C03632=1040.909,-108.162,425.924,168.760,35.372,156.676
C03633=1040.915,-107.912,425.914,168.762,35.372,156.676
C03634=1040.921,-107.663,425.904,168.765,35.371,156.675
C03635=1040.927,-107.413,425.894,168.767,35.371,156.675
C03636=1040.934,-107.163,425.885,168.770,35.371,156.675
C03637=1040.940,-106.913,425.875,168.772,35.371,156.675
C03638=1040.945,-106.663,425.865,168.775,35.370,156.675
C03639=1040.952,-106.414,425.855,168.777,35.370,156.675
C03640=1040.958,-106.164,425.845,168.779,35.370,156.675
C03641=1040.964,-105.914,425.836,168.781,35.370,156.675
C03642=1040.970,-105.665,425.826,168.784,35.370,156.675
C03643=1040.976,-105.414,425.816,168.786,35.369,156.675
C03644=1040.982,-105.165,425.806,168.789,35.369,156.675
C03645=1040.988,-104.915,425.796,168.791,35.369,156.675
C03646=1040.994,-104.666,425.787,168.794,35.369,156.675
C03647=1041.000,-104.416,425.776,168.796,35.369,156.675
C03648=1041.006,-104.166,425.766,168.799,35.368,156.674
C03649=1041.013,-103.917,425.757,168.801,35.368,156.674
C03650=1041.019,-103.667,425.747,168.804,35.368,156.674
C03651=1041.024,-103.417,425.736,168.806,35.368,156.674
C03652=1041.031,-103.168,425.727,168.809,35.368,156.674
C03653=1041.037,-102.918,425.717,168.811,35.367,156.674
C03654=1041.043,-102.668,425.706,168.814,35.368,156.674
C03655=1041.049,-102.418,425.697,168.816,35.368,156.674
C03656=1041.055,-102.169,425.687,168.819,35.367,156.674
C03657=1041.061,-101.919,425.677,168.821,35.367,156.674
C03658=1041.067,-101.669,425.666,168.824,35.367,156.674
C03659=1041.074,-101.419,425.656,168.826,35.367,156.674
C03660=1041.080,-101.170,425.646,168.829,35.367,156.674
C03661=1041.086,-100.920,425.636,168.831,35.367,156.674
C03662=1041.092,-100.670,425.626,168.834,35.366,156.674
C03663=1041.098,-100.421,425.616,168.836,35.366,156.674
C03664=1041.105,-100.134,425.604,168.839,35.366,156.674
C03665=1041.112,-99.846,425.592,168.842,35.366,156.673
C03666=1041.120,-99.559,425.581,168.845,35.366,156.673
C03667=1041.127,-99.272,425.569,168.847,35.366,156.673
C03668=1041.133,-99.022,425.559,168.850,35.365,156.673
C03669=1041.139,-98.772,425.550,168.852,35.365,156.673
C03670=1041.145,-98.523,425.539,168.855,35.366,156.673
C03671=1041.151,-98.273,425.529,168.857,35.366,156.673
C03672=1041.157,-98.024,425.519,168.860,35.365,156.673
C03673=1041.163,-97.773,425.508,168.862,35.365,156.673
C03674=1041.170,-97.524,425.498,168.865,35.365,156.673
C03675=1041.175,-97.274,425.488,168.867,35.365,156.673
C03676=1041.182,-97.025,425.478,168.870,35.365,156.673
C03677=1041.187,-96.775,425.467,168.871,35.365,156.673
C03678=1041.194,-96.525,425.457,168.874,35.365,156.673
C03679=1041.199,-96.276,425.446,168.876,35.365,156.673
C03680=1041.206,-96.025,425.436,168.878,35.365,156.673
C03681=1041.212,-95.776,425.425,168.881,35.365,156.673
C03682=1041.218,-95.526,425.415,168.883,35.365,156.673
C03683=1041.224,-95.277,425.405,168.886,35.365,156.673
C03684=1041.230,-95.027,425.394,168.888,35.365,156.673
C03685=1041.236,-94.778,425.384,168.891,35.365,156.673
C03686=1041.242,-94.527,425.373,168.893,35.365,156.673
C03687=1041.248,-94.278,425.363,168.895,35.365,156.673
C03688=1041.254,-94.028,425.352,168.898,35.366,156.673
C03689=1041.260,-93.778,425.342,168.900,35.365,156.673
C03690=1041.266,-93.529,425.332,168.903,35.365,156.673
C03691=1041.272,-93.279,425.320,168.905,35.365,156.673
C03692=1041.279,-93.029,425.311,168.908,35.365,156.673
C03693=1041.284,-92.780,425.300,168.910,35.365,156.673
C03694=1041.290,-92.530,425.289,168.913,35.365,156.673
C03695=1041.297,-92.280,425.279,168.915,35.365,156.672
C03696=1041.303,-92.030,425.268,168.917,35.366,156.672
C03697=1041.309,-91.781,425.258,168.920,35.366,156.672
C03698=1041.315,-91.531,425.247,168.922,35.366,156.672
C03699=1041.321,-91.281,425.236,168.925,35.366,156.672
C03700=1041.327,-91.031,425.226,168.927,35.366,156.672
C03701=1041.333,-90.782,425.215,168.930,35.366,156.672
C03702=1041.340,-90.533,425.205,168.932,35.366,156.672
C03703=1041.346,-90.283,425.194,168.934,35.366,156.672
C03704=1041.351,-90.033,425.184,168.937,35.366,156.672
C03705=1041.358,-89.783,425.174,168.939,35.366,156.672
C03706=1041.364,-89.533,425.162,168.942,35.366,156.672
C03707=1041.370,-89.284,425.151,168.944,35.366,156.672
C03708=1041.376,-89.034,425.141,168.946,35.366,156.672
C03709=1041.382,-88.785,425.130,168.949,35.366,156.672
C03710=1041.389,-88.535,425.120,168.951,35.367,156.672
C03711=1041.395,-88.285,425.109,168.954,35.367,156.672
C03712=1041.400,-88.036,425.099,168.956,35.367,156.672
C03713=1041.407,-87.786,425.088,168.959,35.367,156.672
C03714=1041.413,-87.536,425.077,168.961,35.367,156.672
C03715=1041.419,-87.287,425.066,168.963,35.367,156.672
C03716=1041.426,-87.037,425.056,168.966,35.367,156.672
C03717=1041.432,-86.787,425.045,168.968,35.367,156.672
C03718=1041.438,-86.537,425.033,168.971,35.367,156.672
C03719=1041.445,-86.288,425.023,168.973,35.367,156.672
C03720=1041.450,-86.038,425.012,168.975,35.367,156.672
C03721=1041.456,-85.788,425.002,168.978,35.367,156.672
C03722=1041.463,-85.538,424.991,168.980,35.367,156.672
C03723=1041.469,-85.289,424.981,168.983,35.367,156.672
C03724=1041.475,-85.039,424.969,168.985,35.368,156.672
C03725=1041.481,-84.790,424.959,168.988,35.368,156.672
C03726=1041.488,-84.539,424.948,168.990,35.368,156.672
C03727=1041.493,-84.290,424.937,168.992,35.368,156.672
C03728=1041.501,-84.005,424.924,168.995,35.369,156.672
C03729=1041.508,-83.721,424.912,168.998,35.369,156.672
C03730=1041.515,-83.435,424.900,169.001,35.369,156.672
C03731=1041.522,-83.151,424.887,169.003,35.369,156.672
C03732=1041.529,-82.901,424.876,169.006,35.369,156.672
C03733=1041.535,-82.652,424.865,169.008,35.369,156.672
C03734=1041.541,-82.402,424.854,169.011,35.369,156.672
C03735=1041.547,-82.152,424.843,169.013,35.369,156.672
C03736=1041.554,-81.902,424.833,169.015,35.369,156.672
C03737=1041.560,-81.653,424.822,169.018,35.369,156.672
C03738=1041.566,-81.403,424.811,169.020,35.370,156.672
C03739=1041.573,-81.153,424.800,169.023,35.370,156.672
C03740=1041.579,-80.903,424.789,169.025,35.370,156.672
C03741=1041.585,-80.654,424.778,169.027,35.370,156.672
C03742=1041.591,-80.403,424.767,169.030,35.370,156.672
C03743=1041.598,-80.155,424.756,169.032,35.370,156.672
C03744=1041.604,-79.905,424.745,169.035,35.370,156.672
C03745=1041.610,-79.655,424.734,169.037,35.370,156.672
C03746=1041.616,-79.405,424.723,169.039,35.371,156.672
C03747=1041.622,-79.156,424.712,169.042,35.371,156.672
C03748=1041.628,-78.905,424.700,169.044,35.371,156.672
C03749=1041.634,-78.656,424.689,169.046,35.372,156.672
C03750=1041.642,-78.407,424.678,169.049,35.372,156.672
C03751=1041.647,-78.157,424.667,169.051,35.372,156.672
C03752=1041.654,-77.907,424.656,169.053,35.372,156.672
C03753=1041.660,-77.658,424.644,169.056,35.373,156.672
C03754=1041.666,-77.408,424.633,169.058,35.373,156.672
C03755=1041.672,-77.158,424.622,169.060,35.373,156.672
C03756=1041.678,-76.909,424.610,169.063,35.374,156.672
C03757=1041.684,-76.659,424.600,169.065,35.374,156.672
C03758=1041.690,-76.409,424.588,169.068,35.374,156.672
C03759=1041.696,-76.160,424.577,169.070,35.375,156.672
C03760=1041.703,-75.910,424.565,169.072,35.375,156.672
C03761=1041.709,-75.661,424.555,169.075,35.375,156.672
C03762=1041.715,-75.410,424.543,169.077,35.375,156.672
C03763=1041.722,-75.161,424.531,169.079,35.376,156.672
C03764=1041.727,-74.911,424.520,169.082,35.376,156.672
C03765=1041.734,-74.661,424.509,169.084,35.376,156.672
C03766=1041.740,-74.412,424.498,169.086,35.376,156.672
C03767=1041.746,-74.162,424.486,169.089,35.376,156.672
C03768=1041.752,-73.913,424.475,169.091,35.377,156.672
C03769=1041.758,-73.663,424.464,169.093,35.377,156.672
C03770=1041.765,-73.413,424.452,169.096,35.378,156.672
C03771=1041.771,-73.164,424.441,169.098,35.378,156.672
C03772=1041.776,-72.913,424.429,169.100,35.379,156.673
C03773=1041.782,-72.665,424.417,169.103,35.379,156.672
C03774=1041.789,-72.414,424.406,169.105,35.380,156.673
C03775=1041.795,-72.166,424.394,169.107,35.380,156.673
C03776=1041.800,-71.915,424.383,169.109,35.380,156.673
C03777=1041.807,-71.665,424.371,169.112,35.380,156.673
C03778=1041.813,-71.416,424.360,169.114,35.381,156.673
C03779=1041.820,-71.166,424.348,169.116,35.381,156.673
C03780=1041.825,-70.917,424.336,169.119,35.382,156.673
C03781=1041.831,-70.667,424.324,169.121,35.382,156.673
C03782=1041.837,-70.417,424.313,169.123,35.383,156.673
C03783=1041.844,-70.168,424.302,169.126,35.383,156.673
C03784=1041.850,-69.918,424.290,169.128,35.383,156.673
C03785=1041.855,-69.669,424.278,169.130,35.384,156.673
C03786=1041.862,-69.419,424.266,169.132,35.384,156.673
C03787=1041.868,-69.169,424.255,169.135,35.385,156.673
C03788=1041.874,-68.920,424.243,169.137,35.385,156.673
C03789=1041.880,-68.669,424.232,169.139,35.386,156.673
C03790=1041.886,-68.420,424.220,169.142,35.386,156.673
C03791=1041.893,-68.171,424.208,169.144,35.386,156.673
C03792=1041.899,-67.888,424.195,169.147,35.387,156.673
C03793=1041.907,-67.605,424.182,169.149,35.387,156.673
C03794=1041.914,-67.323,424.168,169.152,35.388,156.673
C03795=1041.920,-67.040,424.155,169.154,35.389,156.674
C03796=1041.926,-66.790,424.143,169.157,35.389,156.674
C03797=1041.933,-66.540,424.131,169.159,35.390,156.674
C03798=1041.939,-66.291,424.119,169.161,35.390,156.674
C03799=1041.945,-66.042,424.108,169.163,35.390,156.674
C03800=1041.951,-65.791,424.096,169.166,35.390,156.674
C03801=1041.957,-65.542,424.084,169.168,35.391,156.674
C03802=1041.964,-65.293,424.072,169.170,35.392,156.674
C03803=1041.969,-65.042,424.060,169.173,35.392,156.674
C03804=1041.976,-64.793,424.048,169.175,35.393,156.674
C03805=1041.982,-64.544,424.037,169.177,35.393,156.674
C03806=1041.989,-64.294,424.025,169.179,35.393,156.674
C03807=1041.994,-64.044,424.013,169.182,35.394,156.674
C03808=1042.001,-63.794,424.001,169.184,35.394,156.674
C03809=1042.007,-63.545,423.989,169.186,35.395,156.674
C03810=1042.013,-63.295,423.977,169.189,35.395,156.674
C03811=1042.019,-63.045,423.966,169.192,35.396,156.674
C03812=1042.026,-62.796,423.954,169.194,35.396,156.674
C03813=1042.031,-62.546,423.941,169.196,35.396,156.674
C03814=1042.038,-62.297,423.929,169.199,35.397,156.675
C03815=1042.044,-62.047,423.918,169.201,35.398,156.675
C03816=1042.050,-61.797,423.905,169.203,35.398,156.675
C03817=1042.057,-61.547,423.894,169.205,35.399,156.675
C03818=1042.063,-61.298,423.882,169.208,35.399,156.675
C03819=1042.069,-61.049,423.870,169.210,35.399,156.675
C03820=1042.075,-60.799,423.858,169.212,35.400,156.675
C03821=1042.082,-60.549,423.846,169.214,35.400,156.675
C03822=1042.088,-60.300,423.834,169.217,35.401,156.675
C03823=1042.094,-60.050,423.821,169.219,35.402,156.675
C03824=1042.100,-59.800,423.810,169.221,35.402,156.675
C03825=1042.107,-59.551,423.798,169.224,35.402,156.675
C03826=1042.113,-59.301,423.786,169.226,35.403,156.675
C03827=1042.119,-59.051,423.774,169.228,35.403,156.675
C03828=1042.126,-58.802,423.762,169.230,35.404,156.675
C03829=1042.132,-58.552,423.749,169.233,35.405,156.675
C03830=1042.139,-58.302,423.737,169.235,35.405,156.675
C03831=1042.144,-58.053,423.725,169.237,35.405,156.675
C03832=1042.150,-57.804,423.713,169.239,35.406,156.676
C03833=1042.157,-57.554,423.701,169.242,35.406,156.676
C03834=1042.163,-57.304,423.689,169.244,35.407,156.676
C03835=1042.170,-57.055,423.677,169.246,35.407,156.676
C03836=1042.176,-56.805,423.665,169.248,35.408,156.676
C03837=1042.182,-56.555,423.652,169.251,35.408,156.676
C03838=1042.189,-56.306,423.640,169.253,35.409,156.676
C03839=1042.196,-56.056,423.628,169.255,35.409,156.676
C03840=1042.201,-55.806,423.616,169.257,35.410,156.676
C03841=1042.208,-55.556,423.604,169.260,35.410,156.676
C03842=1042.214,-55.308,423.592,169.262,35.410,156.676
C03843=1042.220,-55.058,423.580,169.264,35.411,156.676
C03844=1042.227,-54.808,423.568,169.266,35.412,156.676
C03845=1042.233,-54.558,423.555,169.269,35.412,156.676
C03846=1042.239,-54.309,423.543,169.271,35.413,156.676
C03847=1042.246,-54.059,423.531,169.273,35.413,156.676
C03848=1042.252,-53.809,423.519,169.275,35.414,156.677
C03849=1042.259,-53.560,423.506,169.278,35.414,156.677
C03850=1042.265,-53.310,423.493,169.280,35.415,156.677
C03851=1042.271,-53.061,423.481,169.282,35.416,156.677
C03852=1042.278,-52.811,423.469,169.284,35.416,156.677
C03853=1042.284,-52.561,423.457,169.286,35.416,156.677
C03854=1042.291,-52.312,423.445,169.289,35.417,156.677
C03855=1042.296,-52.062,423.432,169.291,35.417,156.677
C03856=1042.305,-51.781,423.419,169.293,35.418,156.677
C03857=1042.312,-51.499,423.404,169.297,35.419,156.677
C03858=1042.318,-51.218,423.391,169.299,35.419,156.677
C03859=1042.326,-50.937,423.376,169.302,35.420,156.677
C03860=1042.332,-50.687,423.364,169.304,35.420,156.677
C03861=1042.338,-50.437,423.352,169.306,35.421,156.677
C03862=1042.345,-50.188,423.340,169.309,35.421,156.677
C03863=1042.351,-49.938,423.327,169.311,35.422,156.678
C03864=1042.357,-49.688,423.314,169.313,35.423,156.678
C03865=1042.364,-49.439,423.302,169.315,35.424,156.678
C03866=1042.370,-49.189,423.290,169.317,35.424,156.678
C03867=1042.376,-48.940,423.276,169.319,35.425,156.678
C03868=1042.382,-48.690,423.264,169.322,35.426,156.678
C03869=1042.388,-48.440,423.252,169.324,35.426,156.678
C03870=1042.395,-48.191,423.239,169.326,35.427,156.678
C03871=1042.400,-47.941,423.226,169.328,35.428,156.678
C03872=1042.407,-47.692,423.213,169.330,35.428,156.678
C03873=1042.413,-47.442,423.201,169.333,35.429,156.679
C03874=1042.419,-47.192,423.188,169.335,35.430,156.679
C03875=1042.425,-46.943,423.175,169.337,35.431,156.679
C03876=1042.431,-46.693,423.162,169.339,35.431,156.679
C03877=1042.438,-46.444,423.150,169.341,35.432,156.679
C03878=1042.445,-46.194,423.137,169.343,35.433,156.679
C03879=1042.451,-45.944,423.124,169.346,35.433,156.679
C03880=1042.457,-45.695,423.111,169.348,35.434,156.679
C03881=1042.463,-45.445,423.098,169.350,35.435,156.679
C03882=1042.469,-45.195,423.086,169.352,35.435,156.679
C03883=1042.476,-44.946,423.073,169.354,35.436,156.679
C03884=1042.482,-44.696,423.061,169.356,35.436,156.680
C03885=1042.488,-44.447,423.047,169.359,35.437,156.680
C03886=1042.494,-44.197,423.035,169.362,35.438,156.680
C03887=1042.501,-43.948,423.022,169.364,35.438,156.680
C03888=1042.507,-43.698,423.010,169.366,35.439,156.680
C03889=1042.513,-43.449,422.996,169.368,35.440,156.680
C03890=1042.519,-43.198,422.983,169.370,35.440,156.680
C03891=1042.526,-42.949,422.971,169.372,35.441,156.680
C03892=1042.532,-42.699,422.958,169.375,35.442,156.680
C03893=1042.538,-42.450,422.945,169.377,35.443,156.680
C03894=1042.544,-42.200,422.932,169.379,35.443,156.681
C03895=1042.551,-41.951,422.920,169.381,35.444,156.681
C03896=1042.557,-41.701,422.907,169.383,35.445,156.681
C03897=1042.564,-41.451,422.893,169.385,35.445,156.681
C03898=1042.570,-41.202,422.880,169.387,35.446,156.681
C03899=1042.576,-40.952,422.868,169.390,35.447,156.681
C03900=1042.582,-40.703,422.854,169.392,35.447,156.681
C03901=1042.589,-40.453,422.842,169.394,35.448,156.681
C03902=1042.595,-40.204,422.829,169.396,35.449,156.681
C03903=1042.602,-39.954,422.815,169.398,35.450,156.682
C03904=1042.608,-39.704,422.803,169.400,35.451,156.682
C03905=1042.614,-39.455,422.790,169.402,35.452,156.682
C03906=1042.621,-39.205,422.778,169.405,35.452,156.682
C03907=1042.627,-38.956,422.764,169.407,35.453,156.682
C03908=1042.634,-38.706,422.751,169.409,35.454,156.682
C03909=1042.640,-38.456,422.738,169.411,35.454,156.682
C03910=1042.646,-38.207,422.725,169.414,35.455,156.682
C03911=1042.652,-37.958,422.712,169.416,35.456,156.682
C03912=1042.658,-37.708,422.699,169.418,35.456,156.682
C03913=1042.665,-37.458,422.686,169.420,35.458,156.683
C03914=1042.671,-37.209,422.672,169.423,35.459,156.683
C03915=1042.677,-36.959,422.659,169.425,35.459,156.683
C03916=1042.683,-36.710,422.646,169.427,35.460,156.683
C03917=1042.689,-36.460,422.633,169.429,35.461,156.683
C03918=1042.695,-36.210,422.619,169.431,35.461,156.683
C03919=1042.702,-35.961,422.606,169.433,35.463,156.683
C03920=1042.708,-35.680,422.592,169.435,35.463,156.683
C03921=1042.716,-35.399,422.576,169.438,35.464,156.684
C03922=1042.723,-35.118,422.561,169.440,35.465,156.684
C03923=1042.730,-34.837,422.547,169.442,35.466,156.684
C03924=1042.737,-34.587,422.533,169.445,35.467,156.684
C03925=1042.743,-34.338,422.520,169.447,35.467,156.684
C03926=1042.749,-34.088,422.507,169.449,35.469,156.684
C03927=1042.755,-33.839,422.494,169.451,35.469,156.684
C03928=1042.762,-33.589,422.480,169.453,35.470,156.684
C03929=1042.767,-33.340,422.466,169.455,35.471,156.685
C03930=1042.773,-33.090,422.453,169.458,35.472,156.685
C03931=1042.780,-32.840,422.440,169.460,35.473,156.685
C03932=1042.786,-32.591,422.426,169.462,35.474,156.685
C03933=1042.792,-32.341,422.414,169.464,35.474,156.685
C03934=1042.799,-32.092,422.400,169.466,35.475,156.685
C03935=1042.805,-31.842,422.387,169.469,35.476,156.685
C03936=1042.812,-31.593,422.374,169.471,35.477,156.686
C03937=1042.818,-31.343,422.360,169.473,35.478,156.686
C03938=1042.825,-31.093,422.347,169.475,35.478,156.686
C03939=1042.831,-30.844,422.333,169.477,35.479,156.686
C03940=1042.836,-30.595,422.319,169.479,35.480,156.686
C03941=1042.843,-30.345,422.306,169.481,35.481,156.686
C03942=1042.849,-30.095,422.293,169.483,35.482,156.686
C03943=1042.856,-29.846,422.279,169.485,35.483,156.686
C03944=1042.862,-29.596,422.266,169.487,35.483,156.686
C03945=1042.869,-29.347,422.252,169.489,35.484,156.687
C03946=1042.875,-29.098,422.239,169.491,35.485,156.687
C03947=1042.882,-28.848,422.225,169.493,35.486,156.687
C03948=1042.888,-28.598,422.212,169.495,35.487,156.687
C03949=1042.894,-28.348,422.198,169.498,35.487,156.687
C03950=1042.900,-28.099,422.185,169.501,35.489,156.687
C03951=1042.906,-27.850,422.171,169.503,35.489,156.687
C03952=1042.913,-27.600,422.158,169.505,35.490,156.687
C03953=1042.919,-27.350,422.145,169.507,35.491,156.688
C03954=1042.926,-27.100,422.131,169.509,35.491,156.688
C03955=1042.932,-26.851,422.118,169.511,35.493,156.688
C03956=1042.938,-26.602,422.104,169.513,35.493,156.688
C03957=1042.945,-26.352,422.090,169.515,35.494,156.688
C03958=1042.951,-26.102,422.077,169.517,35.495,156.688
C03959=1042.957,-25.853,422.062,169.519,35.496,156.688
C03960=1042.964,-25.603,422.049,169.521,35.497,156.689
C03961=1042.969,-25.354,422.035,169.523,35.498,156.689
C03962=1042.976,-25.104,422.021,169.525,35.499,156.689
C03963=1042.982,-24.855,422.008,169.527,35.500,156.689
C03964=1042.988,-24.605,421.994,169.529,35.501,156.689
C03965=1042.995,-24.356,421.980,169.531,35.502,156.689
C03966=1043.001,-24.106,421.966,169.533,35.503,156.689
C03967=1043.007,-23.856,421.952,169.536,35.504,156.690
C03968=1043.013,-23.607,421.939,169.538,35.505,156.690
C03969=1043.019,-23.358,421.926,169.540,35.506,156.690
C03970=1043.026,-23.108,421.911,169.542,35.506,156.690
C03971=1043.032,-22.859,421.897,169.544,35.508,156.690
C03972=1043.038,-22.608,421.883,169.546,35.508,156.690
C03973=1043.044,-22.359,421.870,169.548,35.510,156.691
C03974=1043.051,-22.110,421.856,169.550,35.510,156.691
C03975=1043.057,-21.860,421.842,169.552,35.511,156.691
C03976=1043.064,-21.610,421.828,169.554,35.512,156.691
C03977=1043.069,-21.361,421.814,169.556,35.513,156.691
C03978=1043.076,-21.112,421.800,169.558,35.514,156.691
C03979=1043.082,-20.862,421.787,169.560,35.515,156.691
C03980=1043.088,-20.612,421.773,169.562,35.516,156.691
C03981=1043.095,-20.363,421.758,169.564,35.517,156.692
C03982=1043.101,-20.114,421.745,169.566,35.518,156.692
C03983=1043.107,-19.864,421.731,169.569,35.519,156.692
C03984=1043.115,-19.582,421.715,169.572,35.520,156.692
C03985=1043.122,-19.301,421.699,169.574,35.521,156.692
C03986=1043.129,-19.018,421.684,169.576,35.522,156.692
C03987=1043.136,-18.737,421.668,169.579,35.523,156.693
C03988=1043.142,-18.487,421.654,169.581,35.524,156.693
C03989=1043.149,-18.238,421.640,169.583,35.525,156.693
C03990=1043.155,-17.988,421.626,169.585,35.526,156.693
C03991=1043.162,-17.739,421.611,169.586,35.527,156.693
C03992=1043.168,-17.489,421.598,169.588,35.528,156.693
C03993=1043.174,-17.239,421.584,169.590,35.529,156.693
C03994=1043.181,-16.990,421.570,169.592,35.530,156.694
C03995=1043.187,-16.740,421.556,169.594,35.531,156.694
C03996=1043.193,-16.491,421.541,169.596,35.531,156.694
C03997=1043.200,-16.241,421.528,169.598,35.533,156.694
C03998=1043.206,-15.993,421.513,169.600,35.533,156.694
C03999=1043.213,-15.743,421.500,169.603,35.535,156.694
C04000=1043.219,-15.492,421.485,169.605,35.535,156.695
C04001=1043.225,-15.244,421.471,169.607,35.536,156.695
C04002=1043.231,-14.993,421.457,169.609,35.537,156.695
C04003=1043.238,-14.745,421.443,169.611,35.539,156.695
C04004=1043.244,-14.495,421.428,169.613,35.539,156.695
C04005=1043.250,-14.245,421.414,169.615,35.541,156.695
C04006=1043.257,-13.996,421.400,169.617,35.541,156.695
C04007=1043.263,-13.746,421.386,169.619,35.543,156.696
C04008=1043.269,-13.497,421.371,169.621,35.543,156.696
C04009=1043.275,-13.247,421.358,169.623,35.545,156.696
C04010=1043.281,-12.998,421.343,169.625,35.545,156.696
C04011=1043.288,-12.748,421.328,169.627,35.547,156.696
C04012=1043.294,-12.498,421.314,169.629,35.548,156.697
C04013=1043.300,-12.249,421.300,169.631,35.549,156.697
C04014=1043.306,-11.999,421.286,169.634,35.550,156.697
C04015=1043.313,-11.750,421.272,169.636,35.551,156.697
C04016=1043.319,-11.501,421.257,169.638,35.552,156.697
C04017=1043.325,-11.251,421.242,169.640,35.553,156.697
C04018=1043.332,-11.002,421.228,169.642,35.554,156.698
C04019=1043.338,-10.752,421.213,169.644,35.555,156.698
C04020=1043.344,-10.503,421.200,169.646,35.556,156.698
C04021=1043.351,-10.253,421.185,169.647,35.557,156.698
C04022=1043.357,-10.004,421.170,169.649,35.558,156.698
C04023=1043.363,-9.754,421.156,169.651,35.559,156.698
C04024=1043.369,-9.504,421.141,169.653,35.560,156.698
C04025=1043.376,-9.255,421.127,169.655,35.561,156.699
C04026=1043.382,-9.006,421.113,169.657,35.562,156.699
C04027=1043.388,-8.756,421.098,169.660,35.563,156.699
C04028=1043.395,-8.507,421.084,169.662,35.564,156.699
C04029=1043.401,-8.258,421.069,169.664,35.565,156.699
C04030=1043.407,-8.007,421.055,169.666,35.567,156.700
C04031=1043.414,-7.758,421.041,169.668,35.567,156.700
C04032=1043.420,-7.509,421.026,169.670,35.569,156.700
C04033=1043.426,-7.259,421.011,169.672,35.569,156.700
C04034=1043.432,-7.009,420.997,169.674,35.571,156.700
C04035=1043.439,-6.760,420.983,169.676,35.571,156.700
C04036=1043.445,-6.511,420.968,169.678,35.573,156.701
C04037=1043.452,-6.261,420.953,169.679,35.574,156.701
C04038=1043.459,-6.012,420.939,169.681,35.575,156.701
C04039=1043.464,-5.762,420.925,169.683,35.576,156.701
C04040=1043.471,-5.513,420.910,169.685,35.577,156.701
C04041=1043.477,-5.263,420.895,169.688,35.578,156.701
C04042=1043.484,-5.014,420.881,169.690,35.579,156.701
C04043=1043.490,-4.765,420.866,169.692,35.580,156.702
C04044=1043.496,-4.515,420.851,169.694,35.581,156.702
C04045=1043.502,-4.265,420.837,169.696,35.582,156.702
C04046=1043.509,-4.015,420.823,169.698,35.583,156.702
C04047=1043.515,-3.766,420.808,169.700,35.584,156.702
C04048=1043.523,-3.483,420.791,169.702,35.585,156.703
C04049=1043.530,-3.199,420.774,169.704,35.587,156.703
C04050=1043.537,-2.915,420.757,169.706,35.588,156.703
C04051=1043.544,-2.633,420.740,169.708,35.589,156.703
C04052=1043.550,-2.384,420.726,169.710,35.590,156.703
C04053=1043.556,-2.134,420.711,169.712,35.591,156.704
C04054=1043.563,-1.884,420.696,169.715,35.592,156.704
C04055=1043.569,-1.635,420.681,169.717,35.594,156.704
C04056=1043.575,-1.386,420.666,169.719,35.595,156.704
C04057=1043.581,-1.136,420.651,169.721,35.596,156.704
C04058=1043.587,-0.886,420.636,169.722,35.597,156.705
C04059=1043.594,-0.637,420.621,169.724,35.598,156.705
C04060=1043.600,-0.388,420.607,169.726,35.600,156.705
C04061=1043.606,-0.138,420.592,169.728,35.600,156.705
C04062=1043.612,0.111,420.577,169.730,35.602,156.705
C04063=1043.619,0.361,420.562,169.732,35.603,156.706
C04064=1043.624,0.610,420.547,169.734,35.604,156.706
C04065=1043.630,0.860,420.532,169.736,35.605,156.706
C04066=1043.637,1.110,420.517,169.738,35.606,156.706
C04067=1043.643,1.359,420.502,169.740,35.608,156.706
C04068=1043.649,1.609,420.487,169.742,35.609,156.706
C04069=1043.655,1.858,420.472,169.744,35.610,156.707
C04070=1043.662,2.107,420.457,169.746,35.611,156.707
C04071=1043.668,2.357,420.442,169.748,35.612,156.707
C04072=1043.675,2.606,420.427,169.750,35.614,156.707
C04073=1043.681,2.856,420.412,169.751,35.614,156.707
C04074=1043.687,3.106,420.397,169.753,35.616,156.708
C04075=1043.693,3.355,420.382,169.755,35.617,156.708
C04076=1043.700,3.604,420.367,169.757,35.618,156.708
C04077=1043.706,3.853,420.352,169.760,35.619,156.708
C04078=1043.713,4.103,420.337,169.762,35.620,156.708
C04079=1043.718,4.353,420.321,169.764,35.621,156.709
C04080=1043.725,4.603,420.306,169.765,35.623,156.709
C04081=1043.731,4.852,420.291,169.767,35.623,156.709
C04082=1043.737,5.101,420.276,169.769,35.625,156.709
C04083=1043.744,5.350,420.261,169.771,35.626,156.709
C04084=1043.750,5.600,420.246,169.773,35.627,156.710
C04085=1043.756,5.850,420.231,169.775,35.628,156.710
C04086=1043.763,6.099,420.216,169.777,35.629,156.710
C04087=1043.769,6.348,420.201,169.778,35.631,156.710
C04088=1043.776,6.598,420.186,169.780,35.632,156.710
C04089=1043.781,6.848,420.170,169.783,35.633,156.710
C04090=1043.788,7.098,420.155,169.785,35.634,156.711
C04091=1043.794,7.346,420.140,169.787,35.635,156.711
C04092=1043.800,7.596,420.125,169.789,35.637,156.711
C04093=1043.807,7.845,420.110,169.791,35.637,156.711
C04094=1043.813,8.094,420.094,169.792,35.639,156.711
C04095=1043.820,8.344,420.079,169.794,35.640,156.712
C04096=1043.826,8.594,420.064,169.796,35.641,156.712
C04097=1043.833,8.843,420.049,169.798,35.642,156.712
C04098=1043.838,9.093,420.033,169.800,35.643,156.712
C04099=1043.845,9.342,420.018,169.802,35.644,156.712
C04100=1043.851,9.591,420.003,169.804,35.646,156.713
C04101=1043.858,9.841,419.988,169.806,35.646,156.713
C04102=1043.864,10.091,419.973,169.808,35.648,156.713
C04103=1043.871,10.340,419.957,169.810,35.649,156.713
C04104=1043.877,10.589,419.942,169.812,35.650,156.713
C04105=1043.884,10.839,419.927,169.814,35.651,156.714
C04106=1043.890,11.088,419.911,169.816,35.652,156.714
C04107=1043.896,11.338,419.896,169.817,35.654,156.714
C04108=1043.903,11.587,419.880,169.819,35.655,156.714
C04109=1043.909,11.837,419.865,169.821,35.656,156.714
C04110=1043.915,12.086,419.850,169.823,35.657,156.714
C04111=1043.922,12.335,419.835,169.825,35.658,156.715
C04112=1043.930,12.620,419.817,169.828,35.660,156.715
C04113=1043.937,12.906,419.800,169.830,35.661,156.715
C04114=1043.944,13.191,419.783,169.832,35.662,156.715
C04115=1043.951,13.476,419.765,169.834,35.663,156.716
C04116=1043.957,13.725,419.749,169.836,35.664,156.716
C04117=1043.964,13.975,419.734,169.838,35.665,156.716
C04118=1043.970,14.224,419.718,169.840,35.667,156.716
C04119=1043.976,14.474,419.703,169.841,35.668,156.716
C04120=1043.983,14.723,419.687,169.843,35.669,156.717
C04121=1043.989,14.973,419.672,169.845,35.671,156.717
C04122=1043.995,15.222,419.656,169.848,35.672,156.717
C04123=1044.001,15.472,419.641,169.850,35.673,156.717
C04124=1044.008,15.721,419.625,169.851,35.674,156.717
C04125=1044.014,15.971,419.609,169.853,35.675,156.718
C04126=1044.021,16.221,419.594,169.855,35.677,156.718
C04127=1044.027,16.470,419.577,169.857,35.678,156.718
C04128=1044.033,16.720,419.563,169.859,35.679,156.718
C04129=1044.040,16.969,419.547,169.860,35.680,156.718
C04130=1044.046,17.219,419.531,169.862,35.682,156.719
C04131=1044.052,17.468,419.516,169.864,35.682,156.719
C04132=1044.058,17.717,419.499,169.866,35.684,156.719
C04133=1044.065,17.967,419.484,169.869,35.685,156.719
C04134=1044.072,18.216,419.469,169.870,35.686,156.719
C04135=1044.077,18.465,419.453,169.872,35.688,156.720
C04136=1044.084,18.715,419.438,169.874,35.689,156.720
C04137=1044.090,18.964,419.421,169.876,35.690,156.720
C04138=1044.096,19.213,419.406,169.878,35.691,156.720
C04139=1044.103,19.463,419.391,169.879,35.692,156.720
C04140=1044.109,19.712,419.374,169.881,35.694,156.721
C04141=1044.116,19.962,419.358,169.883,35.695,156.721
C04142=1044.122,20.211,419.342,169.885,35.696,156.721
C04143=1044.128,20.461,419.327,169.887,35.697,156.721
C04144=1044.134,20.710,419.311,169.889,35.699,156.722
C04145=1044.141,20.959,419.295,169.891,35.700,156.722
C04146=1044.147,21.208,419.279,169.893,35.701,156.722
C04147=1044.153,21.458,419.264,169.895,35.703,156.722
C04148=1044.159,21.707,419.248,169.896,35.704,156.722
C04149=1044.165,21.957,419.232,169.898,35.705,156.723
C04150=1044.172,22.206,419.216,169.900,35.706,156.723
C04151=1044.178,22.457,419.200,169.902,35.707,156.723
C04152=1044.185,22.706,419.184,169.904,35.708,156.723
C04153=1044.191,22.955,419.168,169.905,35.710,156.723
C04154=1044.198,23.204,419.152,169.908,35.711,156.724
C04155=1044.204,23.453,419.136,169.910,35.712,156.724
C04156=1044.209,23.703,419.120,169.912,35.714,156.724
C04157=1044.216,23.952,419.105,169.913,35.715,156.724
C04158=1044.222,24.202,419.089,169.915,35.716,156.725
C04159=1044.229,24.451,419.073,169.917,35.718,156.725
C04160=1044.235,24.701,419.056,169.919,35.719,156.725
C04161=1044.242,24.950,419.041,169.920,35.720,156.725
C04162=1044.248,25.199,419.025,169.922,35.721,156.725
C04163=1044.254,25.448,419.008,169.924,35.723,156.726
C04164=1044.260,25.698,418.993,169.927,35.723,156.726
C04165=1044.267,25.948,418.977,169.929,35.725,156.726
C04166=1044.273,26.197,418.961,169.930,35.726,156.726
C04167=1044.279,26.447,418.945,169.932,35.727,156.726
C04168=1044.286,26.696,418.929,169.934,35.729,156.727
C04169=1044.292,26.945,418.913,169.936,35.730,156.727
C04170=1044.298,27.195,418.896,169.937,35.731,156.727
C04171=1044.305,27.444,418.881,169.939,35.732,156.727
C04172=1044.311,27.693,418.864,169.941,35.734,156.728
C04173=1044.317,27.943,418.848,169.943,35.735,156.728
C04174=1044.324,28.192,418.832,169.945,35.736,156.728
C04175=1044.330,28.442,418.816,169.947,35.738,156.728
C04176=1044.338,28.728,418.797,169.949,35.739,156.729
C04177=1044.345,29.015,418.779,169.951,35.741,156.729
C04178=1044.351,29.302,418.760,169.953,35.742,156.729
C04179=1044.359,29.588,418.741,169.955,35.744,156.729
C04180=1044.365,29.837,418.725,169.957,35.745,156.730
C04181=1044.371,30.086,418.709,169.959,35.746,156.730
C04182=1044.378,30.336,418.693,169.960,35.747,156.730
C04183=1044.384,30.586,418.677,169.963,35.749,156.730
C04184=1044.390,30.835,418.660,169.965,35.750,156.730
C04185=1044.396,31.084,418.644,169.967,35.751,156.731
C04186=1044.402,31.334,418.627,169.968,35.753,156.731
C04187=1044.409,31.583,418.611,169.970,35.754,156.731
C04188=1044.415,31.832,418.595,169.972,35.755,156.731
C04189=1044.421,32.081,418.579,169.973,35.756,156.732
C04190=1044.428,32.331,418.562,169.975,35.758,156.732
C04191=1044.434,32.581,418.546,169.977,35.759,156.732
C04192=1044.440,32.830,418.530,169.980,35.760,156.732
C04193=1044.446,33.079,418.514,169.981,35.762,156.732
C04194=1044.453,33.329,418.496,169.983,35.764,156.733
C04195=1044.459,33.578,418.480,169.985,35.765,156.733
C04196=1044.465,33.827,418.464,169.987,35.766,156.733
C04197=1044.471,34.077,418.448,169.988,35.767,156.733
C04198=1044.478,34.326,418.432,169.990,35.769,156.734
C04199=1044.484,34.576,418.415,169.992,35.770,156.734
C04200=1044.491,34.824,418.398,169.994,35.771,156.734
C04201=1044.497,35.075,418.382,169.996,35.773,156.734
C04202=1044.503,35.324,418.365,169.998,35.774,156.735
C04203=1044.509,35.573,418.349,170.000,35.775,156.735
C04204=1044.517,35.822,418.332,170.002,35.776,156.735
C04205=1044.523,36.072,418.316,170.003,35.778,156.735
C04206=1044.529,36.321,418.300,170.005,35.779,156.735
C04207=1044.535,36.571,418.283,170.007,35.780,156.736
C04208=1044.541,36.820,418.266,170.008,35.782,156.736
C04209=1044.547,37.069,418.250,170.010,35.783,156.736
C04210=1044.555,37.319,418.234,170.013,35.784,156.736
C04211=1044.561,37.568,418.218,170.015,35.786,156.737
C04212=1044.567,37.817,418.201,170.016,35.787,156.737
C04213=1044.573,38.067,418.184,170.018,35.788,156.737
C04214=1044.580,38.316,418.167,170.020,35.789,156.737
C04215=1044.586,38.565,418.151,170.021,35.791,156.738
C04216=1044.592,38.815,418.134,170.023,35.792,156.738
C04217=1044.598,39.064,418.117,170.025,35.793,156.738
C04218=1044.604,39.314,418.101,170.027,35.795,156.738
C04219=1044.610,39.564,418.084,170.029,35.796,156.739
C04220=1044.616,39.812,418.067,170.031,35.798,156.739
C04221=1044.622,40.062,418.051,170.033,35.799,156.739
C04222=1044.629,40.311,418.033,170.034,35.800,156.739
C04223=1044.635,40.560,418.017,170.036,35.802,156.739
C04224=1044.641,40.810,418.001,170.038,35.803,156.740
C04225=1044.648,41.059,417.984,170.040,35.804,156.740
C04226=1044.654,41.309,417.967,170.041,35.805,156.740
C04227=1044.661,41.558,417.950,170.043,35.807,156.740
C04228=1044.667,41.807,417.934,170.046,35.808,156.741
C04229=1044.673,42.056,417.917,170.047,35.810,156.741
C04230=1044.680,42.306,417.900,170.049,35.811,156.741
C04231=1044.686,42.555,417.883,170.051,35.813,156.741
C04232=1044.692,42.804,417.867,170.052,35.814,156.742
C04233=1044.698,43.054,417.849,170.054,35.815,156.742
C04234=1044.704,43.303,417.833,170.056,35.816,156.742
C04235=1044.711,43.553,417.815,170.058,35.818,156.742
C04236=1044.717,43.802,417.799,170.059,35.819,156.742
C04237=1044.723,44.051,417.782,170.062,35.821,156.743
C04238=1044.729,44.301,417.765,170.064,35.822,156.743
C04239=1044.735,44.550,417.748,170.065,35.823,156.743
C04240=1044.742,44.836,417.729,170.067,35.825,156.744
C04241=1044.749,45.123,417.708,170.069,35.827,156.744
C04242=1044.756,45.410,417.689,170.071,35.829,156.744
C04243=1044.763,45.696,417.670,170.073,35.830,156.744
C04244=1044.769,45.946,417.653,170.076,35.832,156.745
C04245=1044.776,46.194,417.636,170.077,35.833,156.745
C04246=1044.782,46.444,417.619,170.079,35.834,156.745
C04247=1044.788,46.693,417.601,170.081,35.836,156.745
C04248=1044.794,46.942,417.584,170.082,35.837,156.746
C04249=1044.801,47.192,417.568,170.084,35.839,156.746
C04250=1044.806,47.441,417.550,170.086,35.840,156.746
C04251=1044.813,47.691,417.533,170.087,35.841,156.746
C04252=1044.819,47.940,417.517,170.089,35.843,156.747
C04253=1044.825,48.190,417.499,170.092,35.844,156.747
C04254=1044.831,48.439,417.482,170.093,35.846,156.747
C04255=1044.838,48.689,417.465,170.095,35.847,156.747
C04256=1044.843,48.938,417.448,170.097,35.848,156.748
C04257=1044.850,49.186,417.431,170.098,35.850,156.748
C04258=1044.856,49.436,417.413,170.100,35.851,156.748
C04259=1044.862,49.685,417.396,170.102,35.853,156.749
C04260=1044.868,49.935,417.379,170.103,35.854,156.749
C04261=1044.874,50.184,417.361,170.106,35.856,156.749
C04262=1044.881,50.434,417.345,170.108,35.857,156.749
C04263=1044.887,50.683,417.328,170.110,35.858,156.749
C04264=1044.893,50.932,417.310,170.111,35.860,156.750
C04265=1044.899,51.181,417.293,170.113,35.861,156.750
C04266=1044.906,51.431,417.276,170.115,35.863,156.750
C04267=1044.911,51.680,417.259,170.116,35.864,156.750
C04268=1044.918,51.930,417.241,170.118,35.865,156.751
C04269=1044.924,52.178,417.224,170.121,35.867,156.751
C04270=1044.930,52.428,417.207,170.122,35.868,156.751
C04271=1044.937,52.677,417.190,170.124,35.870,156.751
C04272=1044.943,52.927,417.173,170.126,35.871,156.752
C04273=1044.949,53.176,417.155,170.127,35.872,156.752
C04274=1044.956,53.425,417.138,170.129,35.873,156.752
C04275=1044.962,53.675,417.120,170.131,35.875,156.753
C04276=1044.968,53.924,417.103,170.132,35.877,156.753
C04277=1044.975,54.173,417.086,170.135,35.878,156.753
C04278=1044.980,54.422,417.068,170.137,35.879,156.753
C04279=1044.987,54.672,417.052,170.138,35.880,156.753
C04280=1044.993,54.921,417.035,170.140,35.882,156.754
C04281=1044.999,55.171,417.017,170.142,35.884,156.754
C04282=1045.006,55.420,416.999,170.143,35.885,156.754
C04283=1045.012,55.669,416.982,170.145,35.886,156.754
C04284=1045.019,55.919,416.964,170.147,35.888,156.755
C04285=1045.025,56.167,416.947,170.149,35.889,156.755
C04286=1045.031,56.417,416.930,170.151,35.890,156.755
C04287=1045.037,56.666,416.913,170.153,35.892,156.755
C04288=1045.043,56.916,416.895,170.154,35.893,156.756
C04289=1045.050,57.165,416.877,170.156,35.895,156.756
C04290=1045.056,57.414,416.860,170.158,35.896,156.756
C04291=1045.063,57.664,416.842,170.160,35.897,156.756
C04292=1045.069,57.913,416.825,170.161,35.898,156.757
C04293=1045.075,58.162,416.807,170.163,35.900,156.757
C04294=1045.082,58.412,416.790,170.166,35.902,156.757
C04295=1045.089,58.661,416.773,170.167,35.903,156.757
C04296=1045.098,59.024,416.748,170.170,35.905,156.758
C04297=1045.107,59.387,416.722,170.172,35.907,156.758
C04298=1045.116,59.749,416.696,170.175,35.909,156.758
C04299=1045.125,60.112,416.671,170.177,35.911,156.759
C04300=1045.136,60.535,416.641,170.181,35.913,156.759
C04301=1045.146,60.956,416.612,170.184,35.915,156.760
C04302=1045.158,61.378,416.583,170.187,35.918,156.760
C04303=1045.169,61.800,416.553,170.189,35.920,156.761
C04304=1045.174,62.049,416.535,170.191,35.921,156.761
C04305=1045.181,62.299,416.518,170.194,35.923,156.761
C04306=1045.187,62.549,416.500,170.196,35.924,156.761
C04307=1045.194,62.797,416.482,170.197,35.925,156.761
C04308=1045.200,63.046,416.464,170.199,35.926,156.762
C04309=1045.207,63.296,416.447,170.201,35.928,156.762
C04310=1045.213,63.545,416.430,170.202,35.929,156.762
C04311=1045.219,63.794,416.412,170.204,35.930,156.762
C04312=1045.226,64.044,416.395,170.206,35.932,156.763
C04313=1045.232,64.293,416.377,170.208,35.933,156.763
C04314=1045.238,64.543,416.358,170.210,35.935,156.763
C04315=1045.244,64.792,416.341,170.212,35.936,156.763
C04316=1045.251,65.041,416.323,170.213,35.938,156.764
C04317=1045.257,65.291,416.305,170.215,35.939,156.764
C04318=1045.263,65.539,416.287,170.217,35.941,156.764
C04319=1045.270,65.789,416.270,170.218,35.942,156.764
C04320=1045.276,66.038,416.252,170.220,35.944,156.765
C04321=1045.282,66.288,416.234,170.223,35.945,156.765
C04322=1045.288,66.536,416.216,170.224,35.946,156.765
C04323=1045.295,66.786,416.198,170.226,35.948,156.765
C04324=1045.301,67.036,416.180,170.228,35.949,156.766
C04325=1045.306,67.284,416.162,170.229,35.951,156.766
C04326=1045.313,67.534,416.145,170.231,35.952,156.766
C04327=1045.319,67.783,416.127,170.233,35.953,156.766
C04328=1045.326,68.032,416.108,170.234,35.955,156.767
C04329=1045.331,68.281,416.091,170.237,35.956,156.767
C04330=1045.338,68.531,416.073,170.239,35.958,156.767
C04331=1045.345,68.780,416.055,170.240,35.959,156.768
C04332=1045.351,69.030,416.037,170.242,35.961,156.768
C04333=1045.356,69.279,416.019,170.244,35.962,156.768
C04334=1045.363,69.528,416.001,170.245,35.963,156.768
C04335=1045.370,69.777,415.983,170.247,35.965,156.769
C04336=1045.376,70.027,415.964,170.250,35.967,156.769
C04337=1045.382,70.276,415.947,170.251,35.968,156.769
C04338=1045.388,70.525,415.929,170.253,35.969,156.769
C04339=1045.394,70.774,415.910,170.254,35.971,156.770
C04340=1045.400,71.024,415.892,170.256,35.972,156.770
C04341=1045.407,71.273,415.874,170.258,35.974,156.770
C04342=1045.413,71.522,415.857,170.259,35.975,156.771
C04343=1045.419,71.771,415.838,170.261,35.977,156.771
C04344=1045.425,72.021,415.820,170.264,35.978,156.771
C04345=1045.432,72.270,415.802,170.265,35.979,156.771
C04346=1045.437,72.519,415.784,170.267,35.981,156.772
C04347=1045.444,72.768,415.765,170.269,35.982,156.772
C04348=1045.450,73.018,415.747,170.270,35.984,156.772
C04349=1045.456,73.267,415.729,170.272,35.986,156.772
C04350=1045.462,73.517,415.711,170.274,35.987,156.773
C04351=1045.468,73.765,415.693,170.276,35.988,156.773
C04352=1045.474,74.015,415.675,170.278,35.990,156.773
C04353=1045.481,74.264,415.656,170.280,35.991,156.773
C04354=1045.488,74.513,415.639,170.281,35.993,156.774
C04355=1045.494,74.763,415.620,170.283,35.995,156.774
C04356=1045.500,75.012,415.602,170.285,35.996,156.774
C04357=1045.506,75.261,415.584,170.286,35.997,156.774
C04358=1045.512,75.510,415.565,170.288,35.998,156.775
C04359=1045.519,75.760,415.547,170.291,36.000,156.775
C04360=1045.525,76.009,415.529,170.292,36.001,156.775
C04361=1045.531,76.258,415.511,170.294,36.003,156.775
C04362=1045.538,76.508,415.492,170.296,36.005,156.776
C04363=1045.544,76.757,415.473,170.297,36.006,156.776
C04364=1045.551,77.043,415.453,170.299,36.007,156.776
C04365=1045.558,77.329,415.432,170.302,36.009,156.777
C04366=1045.565,77.615,415.410,170.304,36.011,156.777
C04367=1045.573,77.901,415.389,170.306,36.012,156.777
C04368=1045.579,78.150,415.371,170.307,36.014,156.778
C04369=1045.585,78.399,415.353,170.309,36.015,156.778
C04370=1045.591,78.648,415.335,170.311,36.017,156.778
C04371=1045.597,78.897,415.315,170.312,36.019,156.778
C04372=1045.603,79.147,415.297,170.315,36.020,156.779
C04373=1045.609,79.396,415.279,170.317,36.022,156.779
C04374=1045.616,79.645,415.260,170.318,36.023,156.779
C04375=1045.622,79.894,415.241,170.320,36.024,156.779
C04376=1045.628,80.144,415.224,170.322,36.026,156.780
C04377=1045.633,80.393,415.205,170.323,36.027,156.780
C04378=1045.640,80.642,415.186,170.325,36.029,156.780
C04379=1045.646,80.891,415.167,170.328,36.031,156.781
C04380=1045.652,81.140,415.149,170.329,36.032,156.781
C04381=1045.659,81.390,415.131,170.331,36.034,156.781
C04382=1045.664,81.639,415.112,170.332,36.035,156.781
C04383=1045.671,81.889,415.093,170.334,36.037,156.782
C04384=1045.677,82.138,415.074,170.336,36.038,156.782
C04385=1045.684,82.387,415.056,170.337,36.039,156.782
C04386=1045.689,82.636,415.038,170.340,36.041,156.783
C04387=1045.695,82.885,415.019,170.342,36.043,156.783
C04388=1045.701,83.134,415.000,170.343,36.044,156.783
C04389=1045.708,83.384,414.981,170.345,36.046,156.783
C04390=1045.714,83.633,414.963,170.347,36.047,156.784
C04391=1045.720,83.882,414.944,170.348,36.049,156.784
C04392=1045.726,84.131,414.925,170.350,36.050,156.784
C04393=1045.733,84.380,414.906,170.353,36.051,156.784
C04394=1045.739,84.630,414.888,170.354,36.053,156.785
C04395=1045.745,84.879,414.870,170.356,36.055,156.785
C04396=1045.751,85.129,414.850,170.358,36.056,156.785
C04397=1045.757,85.378,414.832,170.359,36.058,156.786
C04398=1045.764,85.627,414.813,170.361,36.059,156.786
C04399=1045.770,85.876,414.795,170.363,36.060,156.786
C04400=1045.776,86.125,414.775,170.365,36.062,156.786
C04401=1045.782,86.375,414.757,170.367,36.063,156.787
C04402=1045.789,86.624,414.738,170.369,36.065,156.787
C04403=1045.795,86.873,414.719,170.370,36.067,156.787
C04404=1045.801,87.122,414.700,170.372,36.068,156.787
C04405=1045.807,87.371,414.681,170.374,36.070,156.788
C04406=1045.814,87.620,414.663,170.375,36.071,156.788
C04407=1045.820,87.870,414.644,170.378,36.072,156.788
C04408=1045.826,88.119,414.625,170.380,36.074,156.789
C04409=1045.832,88.368,414.606,170.381,36.075,156.789
C04410=1045.839,88.617,414.588,170.383,36.077,156.789
C04411=1045.845,88.866,414.569,170.385,36.079,156.789
C04412=1045.851,89.116,414.550,170.386,36.080,156.790
C04413=1045.857,89.365,414.531,170.388,36.081,156.790
C04414=1045.864,89.614,414.512,170.391,36.083,156.790
C04415=1045.870,89.863,414.494,170.392,36.084,156.791
C04416=1045.876,90.113,414.475,170.394,36.086,156.791
C04417=1045.882,90.362,414.456,170.396,36.087,156.791
C04418=1045.888,90.611,414.437,170.397,36.089,156.791
C04419=1045.894,90.860,414.418,170.399,36.090,156.792
C04420=1045.901,91.109,414.399,170.401,36.092,156.792
C04421=1045.907,91.358,414.379,170.403,36.093,156.792
C04422=1045.913,91.607,414.361,170.405,36.095,156.792
C04423=1045.919,91.857,414.341,170.406,36.096,156.793
C04424=1045.925,92.106,414.323,170.408,36.098,156.793
C04425=1045.931,92.356,414.303,170.410,36.099,156.793
C04426=1045.937,92.605,414.283,170.411,36.101,156.794
C04427=1045.944,92.854,414.265,170.414,36.103,156.794
C04428=1045.950,93.140,414.243,170.416,36.104,156.794
C04429=1045.958,93.425,414.221,170.418,36.106,156.795
C04430=1045.965,93.712,414.199,170.420,36.108,156.795
C04431=1045.972,93.998,414.176,170.422,36.109,156.795
C04432=1045.978,94.247,414.158,170.423,36.111,156.796
C04433=1045.984,94.496,414.139,170.426,36.113,156.796
C04434=1045.990,94.745,414.120,170.428,36.115,156.796
C04435=1045.996,94.994,414.100,170.429,36.116,156.796
C04436=1046.003,95.243,414.081,170.431,36.118,156.797
C04437=1046.008,95.493,414.062,170.433,36.119,156.797
C04438=1046.015,95.741,414.043,170.434,36.120,156.797
C04439=1046.021,95.991,414.023,170.436,36.122,156.798
C04440=1046.028,96.240,414.004,170.439,36.123,156.798
C04441=1046.033,96.490,413.985,170.440,36.125,156.798
C04442=1046.040,96.738,413.966,170.442,36.126,156.798
C04443=1046.046,96.988,413.947,170.444,36.128,156.799
C04444=1046.052,97.237,413.927,170.445,36.130,156.799
C04445=1046.058,97.486,413.908,170.447,36.131,156.799
C04446=1046.064,97.735,413.889,170.450,36.133,156.800
C04447=1046.070,97.984,413.870,170.451,36.134,156.800
C04448=1046.077,98.234,413.850,170.453,36.136,156.800
C04449=1046.083,98.483,413.831,170.455,36.137,156.800
C04450=1046.089,98.732,413.811,170.456,36.138,156.801
C04451=1046.096,98.981,413.792,170.458,36.140,156.801
C04452=1046.101,99.230,413.773,170.460,36.142,156.801
C04453=1046.107,99.479,413.753,170.462,36.143,156.802
C04454=1046.115,99.729,413.734,170.464,36.145,156.802
C04455=1046.121,99.978,413.714,170.466,36.146,156.802
C04456=1046.127,100.227,413.696,170.468,36.148,156.802
C04457=1046.133,100.476,413.676,170.469,36.149,156.803
C04458=1046.139,100.725,413.656,170.471,36.151,156.803
C04459=1046.145,100.974,413.638,170.473,36.152,156.803
C04460=1046.152,101.224,413.617,170.475,36.154,156.804
C04461=1046.157,101.473,413.598,170.477,36.155,156.804
C04462=1046.163,101.722,413.578,170.479,36.157,156.804
C04463=1046.169,101.971,413.559,170.480,36.159,156.804
C04464=1046.176,102.220,413.540,170.482,36.160,156.805
C04465=1046.181,102.469,413.520,170.484,36.162,156.805
C04466=1046.188,102.719,413.500,170.486,36.164,156.805
C04467=1046.194,102.968,413.480,170.488,36.165,156.806
C04468=1046.200,103.217,413.461,170.490,36.167,156.806
C04469=1046.206,103.466,413.441,170.491,36.169,156.806
C04470=1046.212,103.715,413.422,170.493,36.170,156.806
C04471=1046.218,103.964,413.402,170.495,36.172,156.807
C04472=1046.224,104.214,413.383,170.497,36.173,156.807
C04473=1046.230,104.463,413.363,170.499,36.175,156.807
C04474=1046.236,104.712,413.343,170.501,36.176,156.808
C04475=1046.242,104.961,413.324,170.502,36.178,156.808
C04476=1046.249,105.210,413.304,170.504,36.179,156.808
C04477=1046.255,105.460,413.285,170.506,36.181,156.809
C04478=1046.261,105.709,413.265,170.508,36.182,156.809
C04479=1046.267,105.957,413.245,170.510,36.184,156.809
C04480=1046.273,106.207,413.225,170.512,36.185,156.809
C04481=1046.279,106.456,413.205,170.513,36.187,156.810
C04482=1046.286,106.705,413.186,170.515,36.189,156.810
C04483=1046.292,106.954,413.166,170.517,36.190,156.810
C04484=1046.298,107.203,413.147,170.519,36.192,156.811
C04485=1046.304,107.453,413.126,170.521,36.194,156.811
C04486=1046.310,107.702,413.107,170.523,36.195,156.811
C04487=1046.316,107.951,413.087,170.525,36.197,156.812
C04488=1046.323,108.200,413.067,170.526,36.198,156.812
C04489=1046.329,108.449,413.047,170.528,36.199,156.812
C04490=1046.335,108.698,413.028,170.530,36.201,156.812
C04491=1046.341,108.947,413.008,170.532,36.202,156.813
C04492=1046.348,109.233,412.985,170.534,36.204,156.813
C04493=1046.356,109.519,412.962,170.536,36.206,156.813
C04494=1046.363,109.805,412.940,170.538,36.208,156.814
C04495=1046.370,110.091,412.917,170.540,36.210,156.814
C04496=1046.376,110.340,412.897,170.543,36.211,156.814
C04497=1046.382,110.589,412.877,170.545,36.213,156.815
C04498=1046.389,110.838,412.857,170.546,36.214,156.815
C04499=1046.395,111.087,412.837,170.548,36.216,156.815
C04500=1046.400,111.337,412.818,170.550,36.217,156.815
C04501=1046.407,111.586,412.797,170.551,36.219,156.816
C04502=1046.413,111.835,412.777,170.553,36.221,156.816
C04503=1046.419,112.084,412.757,170.556,36.222,156.816
C04504=1046.425,112.333,412.737,170.557,36.224,156.817
C04505=1046.431,112.582,412.717,170.559,36.226,156.817
C04506=1046.437,112.831,412.697,170.561,36.227,156.817
C04507=1046.444,113.081,412.678,170.563,36.229,156.818
C04508=1046.450,113.330,412.658,170.565,36.231,156.818
C04509=1046.456,113.579,412.638,170.567,36.232,156.818
C04510=1046.462,113.828,412.617,170.569,36.234,156.818
C04511=1046.468,114.077,412.597,170.570,36.235,156.819
C04512=1046.474,114.326,412.577,170.572,36.237,156.819
C04513=1046.480,114.576,412.557,170.574,36.239,156.819
C04514=1046.486,114.824,412.537,170.576,36.240,156.820
C04515=1046.492,115.073,412.517,170.578,36.242,156.820
C04516=1046.497,115.322,412.496,170.580,36.244,156.820
C04517=1046.504,115.572,412.476,170.581,36.245,156.821
C04518=1046.510,115.821,412.456,170.583,36.247,156.821
C04519=1046.515,116.070,412.435,170.585,36.249,156.821
C04520=1046.522,116.319,412.415,170.588,36.250,156.822
C04521=1046.528,116.568,412.395,170.589,36.252,156.822
C04522=1046.534,116.817,412.375,170.591,36.254,156.822
C04523=1046.540,117.067,412.354,170.593,36.255,156.823
C04524=1046.546,117.315,412.333,170.594,36.257,156.823
C04525=1046.552,117.564,412.313,170.596,36.259,156.823
C04526=1046.558,117.814,412.293,170.599,36.260,156.823
C04527=1046.564,118.062,412.273,170.600,36.262,156.824
C04528=1046.570,118.312,412.252,170.602,36.264,156.824
C04529=1046.576,118.561,412.232,170.604,36.265,156.824
C04530=1046.582,118.810,412.212,170.606,36.267,156.825
C04531=1046.588,119.059,412.191,170.608,36.269,156.825
C04532=1046.594,119.308,412.171,170.610,36.270,156.825
C04533=1046.600,119.557,412.150,170.612,36.272,156.826
C04534=1046.606,119.806,412.130,170.613,36.273,156.826
C04535=1046.612,120.055,412.110,170.615,36.275,156.826
C04536=1046.618,120.305,412.089,170.617,36.277,156.827
C04537=1046.624,120.554,412.069,170.620,36.278,156.827
C04538=1046.631,120.803,412.049,170.621,36.280,156.827
C04539=1046.637,121.051,412.028,170.623,36.282,156.828
C04540=1046.642,121.300,412.007,170.625,36.283,156.828
C04541=1046.649,121.550,411.987,170.626,36.285,156.828
C04542=1046.655,121.799,411.967,170.628,36.286,156.828
C04543=1046.661,122.048,411.946,170.631,36.288,156.829
C04544=1046.667,122.297,411.926,170.633,36.290,156.829
C04545=1046.674,122.546,411.905,170.634,36.291,156.829
C04546=1046.679,122.795,411.885,170.636,36.293,156.830
C04547=1046.686,123.044,411.864,170.638,36.295,156.830
C04548=1046.692,123.293,411.844,170.640,36.296,156.830
C04549=1046.698,123.543,411.823,170.642,36.298,156.831
C04550=1046.704,123.792,411.803,170.644,36.299,156.831
C04551=1046.711,124.041,411.782,170.646,36.301,156.831
C04552=1046.716,124.290,411.761,170.648,36.303,156.832
C04553=1046.722,124.539,411.741,170.649,36.304,156.832
C04554=1046.729,124.788,411.720,170.652,36.306,156.832
C04555=1046.735,125.037,411.699,170.654,36.307,156.833
C04556=1046.742,125.323,411.676,170.656,36.309,156.833
C04557=1046.748,125.609,411.653,170.658,36.311,156.833
C04558=1046.755,125.894,411.629,170.660,36.313,156.834
C04559=1046.763,126.180,411.605,170.662,36.315,156.834
C04560=1046.769,126.429,411.585,170.665,36.316,156.834
C04561=1046.775,126.678,411.563,170.666,36.318,156.835
C04562=1046.781,126.927,411.543,170.668,36.320,156.835
C04563=1046.788,127.177,411.523,170.670,36.321,156.835
C04564=1046.793,127.425,411.502,170.672,36.323,156.835
C04565=1046.800,127.675,411.482,170.674,36.325,156.836
C04566=1046.807,127.924,411.461,170.676,36.326,156.836
C04567=1046.812,128.173,411.440,170.678,36.328,156.836
C04568=1046.819,128.422,411.419,170.680,36.330,156.837
C04569=1046.824,128.671,411.398,170.682,36.331,156.837
C04570=1046.831,128.920,411.378,170.683,36.333,156.837
C04571=1046.838,129.169,411.357,170.686,36.335,156.838
C04572=1046.843,129.418,411.336,170.688,36.336,156.838
C04573=1046.850,129.667,411.315,170.690,36.338,156.838
C04574=1046.856,129.916,411.295,170.691,36.339,156.839
C04575=1046.862,130.165,411.274,170.693,36.341,156.839
C04576=1046.869,130.415,411.254,170.695,36.342,156.839
C04577=1046.874,130.663,411.232,170.698,36.344,156.840
C04578=1046.881,130.913,411.212,170.700,36.346,156.840
C04579=1046.887,131.161,411.191,170.701,36.347,156.840
C04580=1046.893,131.411,411.170,170.703,36.349,156.841
C04581=1046.900,131.660,411.149,170.705,36.351,156.841
C04582=1046.905,131.908,411.128,170.708,36.352,156.841
C04583=1046.911,132.158,411.107,170.710,36.354,156.841
C04584=1046.917,132.406,411.086,170.711,36.356,156.842
C04585=1046.923,132.656,411.065,170.713,36.357,156.842
C04586=1046.930,132.905,411.044,170.715,36.359,156.842
C04587=1046.936,133.153,411.023,170.718,36.361,156.843
C04588=1046.942,133.403,411.002,170.719,36.362,156.843
C04589=1046.947,133.652,410.981,170.721,36.364,156.843
C04590=1046.954,133.901,410.960,170.723,36.366,156.844
C04591=1046.960,134.150,410.939,170.725,36.367,156.844
C04592=1046.966,134.399,410.918,170.727,36.369,156.844
C04593=1046.972,134.648,410.897,170.729,36.370,156.845
C04594=1046.978,134.898,410.876,170.731,36.372,156.845
C04595=1046.984,135.146,410.855,170.733,36.374,156.845
C04596=1046.990,135.395,410.833,170.735,36.375,156.846
C04597=1046.997,135.644,410.812,170.736,36.377,156.846
C04598=1047.002,135.893,410.791,170.739,36.379,156.846
C04599=1047.008,136.143,410.770,170.741,36.381,156.847
C04600=1047.015,136.391,410.749,170.743,36.382,156.847
C04601=1047.021,136.640,410.727,170.745,36.384,156.847
C04602=1047.027,136.890,410.706,170.746,36.386,156.848
C04603=1047.034,137.139,410.685,170.749,36.388,156.848
C04604=1047.039,137.387,410.664,170.751,36.389,156.848
C04605=1047.045,137.636,410.642,170.753,36.391,156.849
C04606=1047.051,137.886,410.621,170.755,36.393,156.849
C04607=1047.057,138.134,410.601,170.756,36.395,156.849
C04608=1047.064,138.384,410.579,170.758,36.396,156.850
C04609=1047.070,138.633,410.558,170.761,36.398,156.850
C04610=1047.075,138.881,410.536,170.763,36.400,156.850
C04611=1047.082,139.130,410.515,170.765,36.401,156.851
C04612=1047.088,139.379,410.494,170.767,36.403,156.851
C04613=1047.094,139.629,410.473,170.768,36.405,156.851
C04614=1047.100,139.878,410.451,170.771,36.406,156.852
C04615=1047.106,140.127,410.430,170.773,36.408,156.852
C04616=1047.112,140.376,410.408,170.775,36.409,156.852
C04617=1047.118,140.625,410.387,170.777,36.411,156.853
C04618=1047.124,140.874,410.365,170.778,36.413,156.853
C04619=1047.130,141.123,410.344,170.781,36.415,156.853
C04620=1047.137,141.408,410.319,170.783,36.417,156.854
C04621=1047.144,141.694,410.295,170.785,36.419,156.854
C04622=1047.151,141.979,410.270,170.787,36.421,156.855
C04623=1047.158,142.265,410.246,170.791,36.423,156.855
C04624=1047.164,142.514,410.224,170.792,36.425,156.855
C04625=1047.170,142.763,410.203,170.794,36.427,156.856
C04626=1047.176,143.012,410.181,170.796,36.428,156.856
C04627=1047.182,143.261,410.160,170.798,36.430,156.856
C04628=1047.188,143.510,410.138,170.801,36.432,156.857
C04629=1047.194,143.759,410.117,170.802,36.434,156.857
C04630=1047.201,144.008,410.094,170.804,36.435,156.857
C04631=1047.206,144.256,410.073,170.806,36.437,156.858
C04632=1047.212,144.506,410.051,170.808,36.438,156.858
C04633=1047.219,144.755,410.030,170.811,36.440,156.858
C04634=1047.225,145.004,410.008,170.813,36.442,156.859
C04635=1047.231,145.253,409.986,170.815,36.444,156.859
C04636=1047.236,145.502,409.965,170.816,36.445,156.859
C04637=1047.243,145.751,409.944,170.818,36.447,156.860
C04638=1047.249,146.000,409.922,170.820,36.449,156.860
C04639=1047.255,146.249,409.900,170.823,36.451,156.860
C04640=1047.261,146.498,409.878,170.825,36.453,156.861
C04641=1047.267,146.746,409.857,170.827,36.454,156.861
C04642=1047.274,146.995,409.836,170.829,36.456,156.861
C04643=1047.280,147.244,409.814,170.830,36.458,156.862
C04644=1047.285,147.494,409.792,170.833,36.459,156.862
C04645=1047.292,147.743,409.770,170.835,36.461,156.862
C04646=1047.298,147.992,409.748,170.837,36.463,156.863
C04647=1047.304,148.240,409.727,170.839,36.465,156.863
C04648=1047.310,148.489,409.705,170.842,36.467,156.863
C04649=1047.316,148.739,409.683,170.844,36.468,156.864
C04650=1047.322,148.987,409.661,170.845,36.470,156.864
C04651=1047.329,149.236,409.639,170.847,36.472,156.864
C04652=1047.334,149.486,409.617,170.849,36.474,156.865
C04653=1047.340,149.734,409.596,170.852,36.475,156.865
C04654=1047.346,149.983,409.573,170.854,36.477,156.866
C04655=1047.352,150.232,409.552,170.856,36.479,156.866
C04656=1047.358,150.481,409.530,170.858,36.481,156.866
C04657=1047.365,150.730,409.508,170.859,36.483,156.867
C04658=1047.370,150.980,409.486,170.862,36.485,156.867
C04659=1047.376,151.229,409.464,170.864,36.486,156.867
C04660=1047.382,151.477,409.442,170.866,36.488,156.868
C04661=1047.388,151.726,409.420,170.868,36.490,156.868
C04662=1047.394,151.975,409.398,170.870,36.491,156.868
C04663=1047.400,152.224,409.376,170.873,36.493,156.869
C04664=1047.407,152.473,409.354,170.875,36.495,156.869
C04665=1047.413,152.722,409.332,170.876,36.497,156.869
C04666=1047.419,152.971,409.310,170.878,36.499,156.870
C04667=1047.425,153.221,409.288,170.880,36.501,156.870
C04668=1047.431,153.469,409.266,170.883,36.503,156.871
C04669=1047.437,153.718,409.244,170.885,36.504,156.871
C04670=1047.443,153.966,409.222,170.887,36.506,156.871
C04671=1047.448,154.216,409.200,170.889,36.508,156.872
C04672=1047.455,154.464,409.177,170.892,36.509,156.872
C04673=1047.461,154.713,409.156,170.894,36.511,156.872
C04674=1047.468,154.962,409.133,170.896,36.513,156.873
C04675=1047.473,155.212,409.111,170.897,36.515,156.873
C04676=1047.479,155.460,409.089,170.899,36.517,156.873
C04677=1047.485,155.710,409.067,170.902,36.519,156.874
C04678=1047.491,155.958,409.044,170.904,36.520,156.874
C04679=1047.498,156.207,409.023,170.906,36.522,156.874
C04680=1047.503,156.456,409.000,170.908,36.524,156.875
C04681=1047.509,156.706,408.978,170.910,36.526,156.875
C04682=1047.516,156.954,408.956,170.913,36.528,156.875
C04683=1047.522,157.203,408.933,170.915,36.530,156.876
C04684=1047.528,157.488,408.908,170.917,36.532,156.876
C04685=1047.535,157.774,408.882,170.919,36.534,156.877
C04686=1047.542,158.058,408.857,170.922,36.536,156.877
C04687=1047.549,158.344,408.831,170.924,36.538,156.878
C04688=1047.555,158.593,408.808,170.926,36.540,156.878
C04689=1047.561,158.842,408.787,170.928,36.542,156.878
C04690=1047.568,159.091,408.764,170.931,36.544,156.879
C04691=1047.574,159.340,408.741,170.933,36.546,156.879
C04692=1047.580,159.589,408.720,170.935,36.547,156.879
C04693=1047.585,159.838,408.697,170.937,36.549,156.880
C04694=1047.592,160.086,408.675,170.939,36.551,156.880
C04695=1047.598,160.335,408.652,170.942,36.553,156.880
C04696=1047.604,160.585,408.630,170.944,36.555,156.881
C04697=1047.610,160.833,408.607,170.946,36.557,156.881
C04698=1047.616,161.082,408.585,170.948,36.558,156.882
C04699=1047.622,161.331,408.562,170.951,36.561,156.882
C04700=1047.627,161.580,408.539,170.953,36.563,156.882
C04701=1047.633,161.829,408.517,170.954,36.565,156.883
C04702=1047.639,162.078,408.494,170.956,36.566,156.883
C04703=1047.645,162.327,408.471,170.959,36.568,156.884
C04704=1047.651,162.576,408.448,170.961,36.571,156.884
C04705=1047.657,162.825,408.425,170.963,36.572,156.884
C04706=1047.662,163.074,408.402,170.965,36.574,156.885
C04707=1047.668,163.323,408.381,170.967,36.576,156.885
C04708=1047.674,163.572,408.358,170.970,36.578,156.885
C04709=1047.680,163.821,408.335,170.972,36.580,156.886
C04710=1047.686,164.069,408.312,170.974,36.582,156.886
C04711=1047.691,164.318,408.289,170.976,36.584,156.887
C04712=1047.698,164.567,408.267,170.979,36.586,156.887
C04713=1047.704,164.816,408.244,170.981,36.588,156.887
C04714=1047.709,165.065,408.221,170.983,36.590,156.888
C04715=1047.715,165.314,408.198,170.984,36.592,156.888
C04716=1047.721,165.562,408.175,170.987,36.594,156.889
C04717=1047.727,165.811,408.152,170.989,36.596,156.889
C04718=1047.733,166.060,408.130,170.991,36.598,156.889
C04719=1047.739,166.309,408.107,170.993,36.600,156.890
C04720=1047.744,166.558,408.084,170.996,36.602,156.890
C04721=1047.750,166.807,408.061,170.998,36.604,156.891
C04722=1047.757,167.055,408.038,171.000,36.606,156.891
C04723=1047.762,167.304,408.015,171.002,36.607,156.891
C04724=1047.768,167.553,407.992,171.005,36.610,156.892
C04725=1047.774,167.803,407.969,171.007,36.612,156.892
C04726=1047.780,168.052,407.946,171.009,36.613,156.893
C04727=1047.787,168.300,407.924,171.011,36.615,156.893
C04728=1047.792,168.549,407.901,171.013,36.617,156.893
C04729=1047.798,168.798,407.878,171.016,36.620,156.894
C04730=1047.804,169.047,407.855,171.018,36.621,156.894
C04731=1047.810,169.296,407.832,171.020,36.623,156.895
C04732=1047.816,169.544,407.808,171.022,36.625,156.895
C04733=1047.823,169.793,407.786,171.025,36.627,156.895
C04734=1047.828,170.042,407.763,171.027,36.629,156.896
C04735=1047.834,170.291,407.740,171.029,36.631,156.896
C04736=1047.840,170.540,407.717,171.031,36.633,156.896
C04737=1047.846,170.789,407.694,171.034,36.635,156.897
C04738=1047.852,171.037,407.670,171.036,36.637,156.897
C04739=1047.859,171.286,407.648,171.038,36.639,156.898
C04740=1047.864,171.535,407.625,171.040,36.641,156.898
C04741=1047.870,171.784,407.602,171.043,36.643,156.898
C04742=1047.876,172.033,407.579,171.045,36.645,156.899
C04743=1047.882,172.281,407.555,171.047,36.647,156.899
C04744=1047.888,172.531,407.532,171.049,36.649,156.900
C04745=1047.894,172.780,407.509,171.052,36.651,156.900
C04746=1047.900,173.028,407.486,171.054,36.652,156.900
C04747=1047.906,173.277,407.463,171.056,36.655,156.901
C04748=1047.913,173.562,407.436,171.059,36.657,156.901
C04749=1047.920,173.847,407.410,171.062,36.659,156.902
C04750=1047.927,174.132,407.383,171.064,36.662,156.902
C04751=1047.934,174.417,407.356,171.067,36.663,156.903
C04752=1047.940,174.666,407.334,171.069,36.666,156.903
C04753=1047.946,174.914,407.310,171.072,36.668,156.903
C04754=1047.952,175.163,407.287,171.074,36.670,156.904
C04755=1047.958,175.412,407.264,171.076,36.671,156.904
C04756=1047.965,175.661,407.241,171.078,36.674,156.905
C04757=1047.970,175.910,407.218,171.081,36.676,156.905
C04758=1047.977,176.159,407.194,171.083,36.677,156.905
C04759=1047.983,176.407,407.171,171.085,36.679,156.906
C04760=1047.989,176.656,407.148,171.087,36.682,156.906
C04761=1047.995,176.904,407.125,171.090,36.684,156.907
C04762=1048.001,177.154,407.101,171.092,36.685,156.907
C04763=1048.007,177.403,407.078,171.094,36.687,156.907
C04764=1048.013,177.651,407.055,171.096,36.690,156.908
C04765=1048.020,177.901,407.031,171.099,36.691,156.908
C04766=1048.026,178.149,407.008,171.102,36.693,156.909
C04767=1048.032,178.399,406.984,171.104,36.695,156.909
C04768=1048.038,178.647,406.961,171.106,36.698,156.910
C04769=1048.044,178.896,406.938,171.109,36.699,156.910
C04770=1048.050,179.145,406.914,171.111,36.701,156.910
C04771=1048.057,179.393,406.891,171.113,36.703,156.911
C04772=1048.063,179.642,406.868,171.115,36.705,156.911
C04773=1048.069,179.891,406.844,171.118,36.707,156.911
C04774=1048.075,180.139,406.821,171.120,36.709,156.912
C04775=1048.082,180.389,406.797,171.122,36.711,156.912
C04776=1048.088,180.637,406.774,171.125,36.713,156.913
C04777=1048.093,180.886,406.751,171.128,36.715,156.913
C04778=1048.100,181.135,406.727,171.130,36.717,156.913
C04779=1048.106,181.383,406.703,171.132,36.719,156.914
C04780=1048.112,181.633,406.680,171.134,36.721,156.914
C04781=1048.118,181.881,406.656,171.137,36.723,156.915
C04782=1048.125,182.131,406.633,171.139,36.725,156.915
C04783=1048.131,182.379,406.609,171.141,36.727,156.916
C04784=1048.137,182.627,406.586,171.144,36.729,156.916
C04785=1048.144,182.877,406.563,171.147,36.731,156.916
C04786=1048.150,183.125,406.539,171.149,36.733,156.917
C04787=1048.156,183.374,406.515,171.151,36.735,156.917
C04788=1048.162,183.623,406.492,171.154,36.737,156.918
C04789=1048.169,183.872,406.468,171.156,36.739,156.918
C04790=1048.174,184.120,406.444,171.158,36.741,156.918
C04791=1048.180,184.370,406.421,171.160,36.744,156.919
C04792=1048.186,184.619,406.396,171.164,36.745,156.919
C04793=1048.192,184.867,406.373,171.166,36.748,156.920
C04794=1048.198,185.116,406.349,171.168,36.750,156.920
C04795=1048.204,185.364,406.324,171.170,36.752,156.921
C04796=1048.210,185.613,406.300,171.173,36.754,156.921
C04797=1048.215,185.863,406.277,171.175,36.756,156.921
C04798=1048.221,186.111,406.253,171.177,36.759,156.922
C04799=1048.227,186.360,406.229,171.180,36.761,156.922
C04800=1048.233,186.609,406.205,171.182,36.763,156.923
C04801=1048.239,186.858,406.180,171.185,36.765,156.923
C04802=1048.245,187.106,406.157,171.187,36.767,156.924
C04803=1048.251,187.355,406.132,171.190,36.770,156.924
C04804=1048.257,187.604,406.108,171.192,36.772,156.925
C04805=1048.263,187.852,406.084,171.194,36.774,156.925
C04806=1048.269,188.101,406.060,171.197,36.776,156.925
C04807=1048.274,188.350,406.036,171.199,36.778,156.926
C04808=1048.281,188.599,406.012,171.202,36.781,156.926
C04809=1048.286,188.847,405.987,171.204,36.782,156.927
C04810=1048.293,189.096,405.963,171.207,36.785,156.927
C04811=1048.298,189.345,405.939,171.209,36.787,156.928
C04812=1048.305,189.630,405.912,171.211,36.790,156.928
C04813=1048.312,189.913,405.884,171.215,36.792,156.929
C04814=1048.319,190.198,405.857,171.217,36.795,156.929
C04815=1048.326,190.483,405.829,171.220,36.797,156.930
C04816=1048.332,190.732,405.805,171.223,36.799,156.930
C04817=1048.339,190.980,405.780,171.225,36.801,156.931
C04818=1048.344,191.229,405.756,171.227,36.804,156.931
C04819=1048.350,191.477,405.732,171.230,36.806,156.932
C04820=1048.356,191.726,405.708,171.233,36.808,156.932
C04821=1048.362,191.975,405.684,171.235,36.810,156.933
C04822=1048.368,192.224,405.660,171.237,36.813,156.933
C04823=1048.374,192.473,405.635,171.240,36.814,156.933
C04824=1048.380,192.721,405.611,171.243,36.817,156.934
C04825=1048.386,192.970,405.586,171.245,36.819,156.934
C04826=1048.392,193.219,405.562,171.247,36.821,156.935
C04827=1048.398,193.467,405.538,171.250,36.823,156.935
C04828=1048.404,193.716,405.514,171.252,36.826,156.936
C04829=1048.410,193.965,405.489,171.255,36.828,156.936
C04830=1048.417,194.213,405.465,171.258,36.830,156.937
C04831=1048.423,194.463,405.440,171.260,36.833,156.937
C04832=1048.429,194.711,405.416,171.262,36.834,156.938
C04833=1048.434,194.960,405.392,171.265,36.837,156.938
C04834=1048.441,195.208,405.367,171.268,36.839,156.939
C04835=1048.447,195.457,405.343,171.270,36.841,156.939
C04836=1048.453,195.706,405.318,171.272,36.843,156.939
C04837=1048.459,195.955,405.294,171.275,36.846,156.940
C04838=1048.465,196.203,405.269,171.278,36.848,156.940
C04839=1048.472,196.452,405.245,171.280,36.850,156.941
C04840=1048.477,196.701,405.221,171.283,36.852,156.941
C04841=1048.484,196.949,405.196,171.285,36.855,156.942
C04842=1048.490,197.199,405.171,171.288,36.857,156.942
C04843=1048.495,197.447,405.147,171.291,36.859,156.943
C04844=1048.502,197.696,405.122,171.293,36.861,156.943
C04845=1048.508,197.945,405.098,171.295,36.863,156.944
C04846=1048.514,198.194,405.074,171.298,36.866,156.944
C04847=1048.520,198.442,405.049,171.301,36.868,156.945
C04848=1048.527,198.691,405.025,171.303,36.870,156.945
C04849=1048.533,198.939,405.000,171.305,36.872,156.945
C04850=1048.538,199.188,404.975,171.309,36.875,156.946
C04851=1048.545,199.436,404.951,171.311,36.877,156.946
C04852=1048.551,199.686,404.926,171.313,36.879,156.947
C04853=1048.558,199.935,404.902,171.316,36.881,156.947
C04854=1048.564,200.183,404.877,171.319,36.884,156.948
C04855=1048.569,200.432,404.852,171.321,36.886,156.948
C04856=1048.576,200.680,404.828,171.323,36.888,156.949
C04857=1048.582,200.930,404.803,171.327,36.890,156.949
C04858=1048.589,201.178,404.778,171.329,36.893,156.950
C04859=1048.595,201.426,404.753,171.331,36.895,156.950
C04860=1048.600,201.675,404.729,171.335,36.898,156.951
C04861=1048.607,201.924,404.703,171.337,36.900,156.951
C04862=1048.613,202.173,404.679,171.339,36.902,156.952
C04863=1048.618,202.421,404.654,171.342,36.904,156.952
C04864=1048.624,202.670,404.628,171.345,36.907,156.953
C04865=1048.631,202.919,404.604,171.347,36.909,156.953
C04866=1048.637,203.167,404.579,171.350,36.911,156.954
C04867=1048.643,203.416,404.554,171.352,36.914,156.954
C04868=1048.649,203.665,404.529,171.355,36.916,156.955
C04869=1048.655,203.913,404.504,171.358,36.919,156.955
C04870=1048.661,204.162,404.479,171.360,36.921,156.956
C04871=1048.667,204.411,404.454,171.363,36.923,156.956
C04872=1048.673,204.659,404.429,171.366,36.926,156.957
C04873=1048.679,204.908,404.404,171.368,36.928,156.957
C04874=1048.685,205.157,404.378,171.371,36.931,156.958
C04875=1048.691,205.406,404.354,171.374,36.933,156.958
C04876=1048.717,206.458,404.248,171.612,37.031,156.979
C04877=1048.724,206.719,404.220,171.614,37.034,156.980
C04878=1048.731,206.980,404.193,171.616,37.038,156.981
C04879=1048.738,207.241,404.165,171.618,37.041,156.981
C04880=1048.744,207.502,404.137,171.621,37.044,156.982
C04881=1048.751,207.750,404.111,171.622,37.047,156.983
C04882=1048.758,207.999,404.086,171.625,37.051,156.984
C04883=1048.763,208.248,404.059,171.626,37.054,156.984
C04884=1048.770,208.496,404.033,171.628,37.057,156.985
C04885=1048.777,208.744,404.007,171.631,37.060,156.986
C04886=1048.783,208.992,403.981,171.632,37.063,156.986
C04887=1048.790,209.242,403.954,171.635,37.066,156.987
C04888=1048.796,209.490,403.928,171.636,37.069,156.988
C04889=1048.803,209.739,403.902,171.639,37.073,156.988
C04890=1048.809,209.987,403.875,171.640,37.076,156.989
C04891=1048.815,210.235,403.849,171.643,37.079,156.990
C04892=1048.822,210.484,403.822,171.645,37.082,156.990
C04893=1048.828,210.732,403.796,171.647,37.085,156.991
C04894=1048.835,210.982,403.770,171.649,37.088,156.992
C04895=1048.841,211.230,403.744,171.650,37.092,156.992
C04896=1048.848,211.479,403.717,171.653,37.095,156.993
C04897=1048.855,211.727,403.691,171.655,37.098,156.994
C04898=1048.861,211.976,403.664,171.657,37.101,156.994
C04899=1048.867,212.224,403.638,171.659,37.105,156.995
C04900=1048.873,212.472,403.611,171.661,37.108,156.996
C04901=1048.880,212.721,403.585,171.663,37.110,156.996
C04902=1048.886,212.970,403.558,171.666,37.114,156.997
C04903=1048.892,213.219,403.531,171.667,37.117,156.998
C04904=1048.899,213.467,403.505,171.670,37.120,156.998
C04905=1048.905,213.716,403.478,171.671,37.124,156.999
C04906=1048.912,213.964,403.452,171.673,37.127,157.000
C04907=1048.918,214.213,403.425,171.676,37.130,157.000
C04908=1048.925,214.461,403.399,171.677,37.133,157.001
C04909=1048.931,214.709,403.372,171.680,37.136,157.002
C04910=1048.938,214.957,403.345,171.682,37.139,157.002
C04911=1048.944,215.206,403.319,171.684,37.143,157.003
C04912=1048.950,215.455,403.292,171.686,37.146,157.004
C04913=1048.957,215.703,403.266,171.688,37.149,157.004
C04914=1048.963,215.952,403.239,171.690,37.152,157.005
C04915=1048.970,216.200,403.213,171.693,37.155,157.006
C04916=1048.976,216.449,403.186,171.694,37.158,157.006
C04917=1048.983,216.697,403.158,171.697,37.161,157.007
C04918=1048.989,216.945,403.132,171.699,37.165,157.008
C04919=1048.995,217.195,403.105,171.701,37.168,157.008
C04920=1049.002,217.443,403.079,171.703,37.171,157.009
C04921=1049.008,217.692,403.052,171.705,37.174,157.010
C04922=1049.015,217.939,403.025,171.707,37.177,157.010
C04923=1049.022,218.188,402.998,171.709,37.180,157.011
C04924=1049.028,218.436,402.972,171.712,37.183,157.012
C04925=1049.034,218.685,402.945,171.713,37.186,157.012
C04926=1049.041,218.934,402.917,171.716,37.189,157.013
C04927=1049.048,219.182,402.891,171.718,37.193,157.014
C04928=1049.054,219.431,402.864,171.721,37.196,157.014
C04929=1049.061,219.679,402.838,171.722,37.199,157.015
C04930=1049.067,219.927,402.810,171.725,37.202,157.016
C04931=1049.074,220.176,402.783,171.727,37.205,157.016
C04932=1049.080,220.424,402.757,171.729,37.208,157.017
C04933=1049.087,220.691,402.727,171.731,37.211,157.018
C04934=1049.094,220.958,402.699,171.734,37.215,157.018
C04935=1049.101,221.224,402.670,171.736,37.218,157.019
C04936=1049.107,221.491,402.640,171.738,37.221,157.020
C04937=1049.114,221.740,402.613,171.740,37.225,157.021
C04938=1049.120,221.988,402.587,171.742,37.228,157.021
C04939=1049.127,222.236,402.560,171.745,37.231,157.022
C04940=1049.133,222.485,402.533,171.746,37.234,157.023
C04941=1049.139,222.733,402.505,171.749,37.237,157.023
C04942=1049.146,222.982,402.478,171.751,37.240,157.024
C04943=1049.152,223.230,402.451,171.754,37.243,157.025
C04944=1049.158,223.479,402.424,171.755,37.246,157.025
C04945=1049.166,223.727,402.397,171.758,37.250,157.026
C04946=1049.171,223.975,402.370,171.760,37.253,157.027
C04947=1049.178,224.224,402.342,171.763,37.256,157.027
C04948=1049.184,224.473,402.315,171.764,37.259,157.028
C04949=1049.191,224.720,402.288,171.767,37.262,157.029
C04950=1049.197,224.970,402.261,171.769,37.265,157.029
C04951=1049.204,225.218,402.233,171.772,37.268,157.030
C04952=1049.210,225.466,402.206,171.773,37.271,157.031
C04953=1049.217,225.714,402.179,171.776,37.275,157.031
C04954=1049.223,225.963,402.152,171.778,37.278,157.032
C04955=1049.229,226.211,402.125,171.780,37.281,157.033
C04956=1049.236,226.460,402.097,171.782,37.284,157.033
C04957=1049.243,226.708,402.070,171.784,37.287,157.034
C04958=1049.249,226.957,402.043,171.787,37.290,157.035
C04959=1049.255,227.205,402.015,171.789,37.293,157.035
C04960=1049.261,227.454,401.988,171.791,37.296,157.036
C04961=1049.269,227.702,401.961,171.793,37.299,157.037
C04962=1049.276,227.951,401.933,171.796,37.302,157.037
C04963=1049.282,228.198,401.906,171.798,37.306,157.038
C04964=1049.288,228.447,401.879,171.801,37.309,157.039
C04965=1049.295,228.696,401.851,171.802,37.312,157.039
C04966=1049.301,228.944,401.823,171.805,37.314,157.040
C04967=1049.307,229.193,401.797,171.807,37.317,157.041
C04968=1049.314,229.441,401.769,171.810,37.321,157.041
C04969=1049.320,229.690,401.741,171.812,37.324,157.042
C04970=1049.327,229.938,401.714,171.814,37.327,157.043
C04971=1049.332,230.186,401.686,171.816,37.330,157.043
C04972=1049.339,230.435,401.659,171.819,37.333,157.044
C04973=1049.346,230.684,401.631,171.821,37.336,157.045
C04974=1049.352,230.932,401.603,171.823,37.339,157.045
C04975=1049.358,231.180,401.576,171.825,37.342,157.046
C04976=1049.365,231.428,401.548,171.827,37.345,157.047
C04977=1049.372,231.677,401.520,171.830,37.349,157.047
C04978=1049.378,231.925,401.493,171.832,37.352,157.048
C04979=1049.385,232.173,401.465,171.835,37.355,157.049
C04980=1049.390,232.422,401.438,171.837,37.358,157.049
C04981=1049.397,232.671,401.410,171.839,37.361,157.050
C04982=1049.403,232.919,401.382,171.841,37.364,157.051
C04983=1049.410,233.167,401.354,171.844,37.367,157.051
C04984=1049.416,233.416,401.326,171.846,37.370,157.052
C04985=1049.422,233.664,401.299,171.849,37.374,157.053
C04986=1049.429,233.912,401.271,171.851,37.377,157.053
C04987=1049.436,234.161,401.243,171.853,37.380,157.054
C04988=1049.441,234.410,401.215,171.855,37.383,157.055
C04989=1049.448,234.668,401.186,171.858,37.386,157.055
C04990=1049.455,234.927,401.157,171.860,37.389,157.056
C04991=1049.462,235.186,401.128,171.863,37.393,157.057
C04992=1049.468,235.446,401.099,171.865,37.395,157.058
C04993=1049.475,235.693,401.071,171.868,37.398,157.058
C04994=1049.481,235.942,401.042,171.870,37.402,157.059
C04995=1049.488,236.191,401.015,171.873,37.405,157.060
C04996=1049.495,236.439,400.987,171.874,37.408,157.060
C04997=1049.500,236.687,400.959,171.877,37.411,157.061
C04998=1049.507,236.936,400.931,171.879,37.414,157.062
C04999=1049.513,237.184,400.904,171.882,37.417,157.062
C05000=1049.520,237.432,400.876,171.884,37.420,157.063
C05001=1049.526,237.681,400.847,171.887,37.423,157.064
C05002=1049.533,237.929,400.819,171.889,37.426,157.064
C05003=1049.540,238.177,400.791,171.892,37.429,157.065
C05004=1049.546,238.426,400.763,171.894,37.433,157.066
C05005=1049.552,238.675,400.735,171.897,37.436,157.066
C05006=1049.559,238.922,400.707,171.898,37.439,157.067
C05007=1049.565,239.171,400.679,171.901,37.441,157.068
C05008=1049.571,239.419,400.651,171.903,37.444,157.068
C05009=1049.578,239.667,400.623,171.906,37.448,157.069
C05010=1049.584,239.916,400.594,171.908,37.451,157.070
C05011=1049.591,240.164,400.567,171.911,37.454,157.070
C05012=1049.598,240.412,400.539,171.913,37.457,157.071
C05013=1049.604,240.661,400.510,171.916,37.460,157.072
C05014=1049.611,240.909,400.482,171.918,37.463,157.072
C05015=1049.617,241.158,400.454,171.921,37.466,157.073
C05016=1049.624,241.406,400.425,171.923,37.469,157.074
C05017=1049.630,241.654,400.398,171.926,37.472,157.074
C05018=1049.636,241.903,400.369,171.928,37.475,157.075
C05019=1049.642,242.151,400.340,171.931,37.479,157.076
C05020=1049.649,242.399,400.313,171.932,37.482,157.076
C05021=1049.655,242.647,400.284,171.935,37.484,157.077
C05022=1049.662,242.896,400.256,171.937,37.487,157.078
C05023=1049.668,243.144,400.227,171.940,37.491,157.078
C05024=1049.674,243.393,400.198,171.942,37.494,157.079
C05025=1049.681,243.641,400.170,171.945,37.497,157.080
C05026=1049.687,243.889,400.142,171.947,37.500,157.081
C05027=1049.694,244.137,400.113,171.950,37.503,157.081
C05028=1049.700,244.386,400.085,171.952,37.506,157.082
C05029=1049.706,244.634,400.056,171.955,37.509,157.083
C05030=1049.713,244.883,400.028,171.957,37.513,157.083
C05031=1049.719,245.131,399.999,171.960,37.516,157.084
C05032=1049.726,245.379,399.971,171.962,37.519,157.085
C05033=1049.732,245.627,399.942,171.965,37.521,157.085
C05034=1049.738,245.875,399.913,171.967,37.524,157.086
C05035=1049.744,246.124,399.885,171.970,37.528,157.087
C05036=1049.751,246.372,399.857,171.972,37.531,157.087
C05037=1049.758,246.620,399.827,171.975,37.534,157.088
C05038=1049.764,246.869,399.799,171.977,37.537,157.089
C05039=1049.770,247.117,399.770,171.980,37.540,157.089
C05040=1049.776,247.365,399.741,171.982,37.544,157.090
C05041=1049.782,247.614,399.713,171.985,37.547,157.091
C05042=1049.789,247.862,399.684,171.987,37.550,157.091
C05043=1049.795,248.110,399.655,171.990,37.553,157.092
C05044=1049.801,248.358,399.626,171.992,37.556,157.093
C05045=1049.808,248.611,399.597,171.995,37.559,157.094
C05046=1049.814,248.865,399.567,171.997,37.563,157.094
C05047=1049.821,249.118,399.538,172.000,37.565,157.095
C05048=1049.827,249.372,399.509,172.002,37.569,157.096
C05049=1049.833,249.620,399.480,172.005,37.572,157.096
C05050=1049.840,249.868,399.451,172.007,37.575,157.097
C05051=1049.846,250.116,399.421,172.010,37.578,157.098
C05052=1049.853,250.364,399.393,172.012,37.581,157.099
C05053=1049.859,250.613,399.365,172.015,37.584,157.099
C05054=1049.865,250.861,399.336,172.017,37.587,157.100
C05055=1049.872,251.109,399.306,172.020,37.591,157.101
C05056=1049.878,251.358,399.277,172.022,37.594,157.101
C05057=1049.884,251.606,399.248,172.025,37.596,157.102
C05058=1049.891,251.854,399.219,172.028,37.600,157.103
C05059=1049.897,252.102,399.190,172.030,37.603,157.103
C05060=1049.903,252.350,399.161,172.033,37.606,157.104
C05061=1049.910,252.598,399.133,172.036,37.609,157.105
C05062=1049.917,252.847,399.103,172.039,37.612,157.105
C05063=1049.923,253.095,399.074,172.041,37.615,157.106
C05064=1049.930,253.343,399.045,172.044,37.618,157.107
C05065=1049.936,253.591,399.016,172.046,37.621,157.107
C05066=1049.942,253.839,398.987,172.049,37.625,157.108
C05067=1049.949,254.088,398.958,172.051,37.627,157.109
C05068=1049.955,254.336,398.929,172.054,37.630,157.109
C05069=1049.961,254.584,398.900,172.056,37.634,157.110
C05070=1049.968,254.833,398.871,172.059,37.637,157.111
C05071=1049.974,255.081,398.841,172.061,37.640,157.112
C05072=1049.981,255.329,398.813,172.064,37.643,157.112
C05073=1049.988,255.577,398.784,172.067,37.646,157.113
C05074=1049.994,255.825,398.755,172.070,37.649,157.114
C05075=1050.000,256.074,398.726,172.072,37.652,157.114
C05076=1050.007,256.322,398.695,172.075,37.655,157.115
C05077=1050.014,256.570,398.666,172.077,37.658,157.116
C05078=1050.020,256.818,398.637,172.080,37.661,157.116
C05079=1050.027,257.067,398.608,172.082,37.664,157.117
C05080=1050.033,257.315,398.579,172.085,37.667,157.118
C05081=1050.039,257.563,398.550,172.088,37.671,157.119
C05082=1050.046,257.811,398.520,172.091,37.673,157.119
C05083=1050.053,258.060,398.491,172.093,37.676,157.120
C05084=1050.059,258.308,398.462,172.096,37.679,157.120
C05085=1050.065,258.556,398.433,172.098,37.682,157.121
C05086=1050.072,258.804,398.403,172.101,37.686,157.122
C05087=1050.079,259.052,398.373,172.105,37.689,157.123
C05088=1050.085,259.300,398.344,172.107,37.692,157.123
C05089=1050.092,259.549,398.315,172.110,37.694,157.124
C05090=1050.098,259.797,398.285,172.112,37.698,157.125
C05091=1050.106,260.045,398.256,172.115,37.701,157.125
C05092=1050.112,260.293,398.227,172.117,37.704,157.126
C05093=1050.119,260.541,398.198,172.121,37.707,157.127
C05094=1050.125,260.790,398.168,172.123,37.710,157.127
C05095=1050.132,261.038,398.139,172.126,37.713,157.128
C05096=1050.139,261.286,398.109,172.128,37.716,157.129
C05097=1050.145,261.534,398.080,172.131,37.719,157.129
C05098=1050.152,261.782,398.050,172.134,37.722,157.130
C05099=1050.159,262.030,398.021,172.137,37.725,157.131
C05100=1050.165,262.278,397.991,172.139,37.728,157.132
C05101=1050.171,262.530,397.961,172.142,37.731,157.132
C05102=1050.178,262.781,397.931,172.144,37.734,157.133
C05103=1050.184,263.033,397.901,172.148,37.737,157.134
C05104=1050.191,263.285,397.871,172.151,37.740,157.134
C05105=1050.198,263.533,397.841,172.153,37.744,157.135
C05106=1050.204,263.781,397.812,172.156,37.747,157.136
C05107=1050.211,264.030,397.781,172.159,37.750,157.137
C05108=1050.217,264.278,397.752,172.162,37.753,157.137
C05109=1050.223,264.525,397.722,172.164,37.756,157.138
C05110=1050.230,264.774,397.692,172.167,37.759,157.139
C05111=1050.236,265.022,397.663,172.169,37.762,157.139
C05112=1050.243,265.270,397.632,172.173,37.765,157.140
C05113=1050.249,265.518,397.602,172.176,37.769,157.141
C05114=1050.255,265.767,397.572,172.178,37.772,157.141
C05115=1050.262,266.015,397.543,172.181,37.775,157.142
C05116=1050.268,266.262,397.513,172.184,37.778,157.143
C05117=1050.275,266.511,397.483,172.187,37.781,157.144
C05118=1050.281,266.759,397.453,172.189,37.784,157.144
C05119=1050.288,267.007,397.423,172.192,37.787,157.145
C05120=1050.294,267.255,397.393,172.194,37.790,157.146
C05121=1050.301,267.504,397.363,172.198,37.794,157.146
C05122=1050.308,267.751,397.333,172.200,37.797,157.147
C05123=1050.314,268.000,397.303,172.203,37.799,157.148
C05124=1050.320,268.247,397.273,172.207,37.803,157.149
C05125=1050.327,268.496,397.242,172.209,37.806,157.149
C05126=1050.333,268.743,397.213,172.212,37.809,157.150
C05127=1050.340,268.992,397.183,172.214,37.812,157.151
C05128=1050.346,269.240,397.153,172.218,37.816,157.152
C05129=1050.353,269.488,397.122,172.220,37.819,157.152
C05130=1050.359,269.736,397.092,172.223,37.821,157.153
C05131=1050.366,269.984,397.062,172.225,37.825,157.154
C05132=1050.372,270.232,397.032,172.229,37.828,157.154
C05133=1050.378,270.480,397.001,172.232,37.831,157.155
C05134=1050.385,270.728,396.971,172.234,37.834,157.156
C05135=1050.391,270.976,396.941,172.238,37.837,157.156
C05136=1050.399,271.225,396.911,172.240,37.840,157.157
C05137=1050.404,271.472,396.880,172.243,37.843,157.158
C05138=1050.412,271.721,396.850,172.246,37.847,157.159
C05139=1050.417,271.968,396.820,172.249,37.850,157.159
C05140=1050.425,272.217,396.790,172.252,37.853,157.160
C05141=1050.430,272.464,396.759,172.254,37.856,157.161
C05142=1050.437,272.713,396.729,172.258,37.860,157.162
C05143=1050.444,272.961,396.698,172.260,37.862,157.162
C05144=1050.450,273.209,396.668,172.263,37.866,157.163
C05145=1050.456,273.458,396.637,172.266,37.869,157.164
C05146=1050.463,273.704,396.607,172.269,37.872,157.165
C05147=1050.469,273.953,396.576,172.272,37.875,157.165
C05148=1050.475,274.201,396.546,172.275,37.879,157.166
C05149=1050.482,274.449,396.516,172.278,37.881,157.167
C05150=1050.489,274.698,396.485,172.280,37.885,157.167
C05151=1050.495,274.945,396.454,172.284,37.888,157.168
C05152=1050.502,275.193,396.424,172.286,37.891,157.169
C05153=1050.509,275.441,396.393,172.289,37.894,157.170
C05154=1050.514,275.689,396.363,172.293,37.898,157.170
C05155=1050.521,275.937,396.331,172.295,37.900,157.171
C05156=1050.528,276.186,396.301,172.298,37.904,157.172
C05157=1050.534,276.441,396.270,172.301,37.907,157.173
C05158=1050.541,276.697,396.238,172.304,37.910,157.173
C05159=1050.547,276.953,396.206,172.308,37.914,157.174
C05160=1050.555,277.209,396.175,172.310,37.917,157.175
C05161=1050.561,277.457,396.144,172.314,37.920,157.176
C05162=1050.567,277.705,396.113,172.316,37.923,157.176
C05163=1050.574,277.953,396.082,172.319,37.926,157.177
C05164=1050.580,278.201,396.052,172.323,37.930,157.178
C05165=1050.587,278.449,396.021,172.325,37.933,157.179
C05166=1050.594,278.697,395.990,172.329,37.936,157.179
C05167=1050.599,278.945,395.959,172.331,37.939,157.180
C05168=1050.606,279.193,395.928,172.334,37.942,157.181
C05169=1050.613,279.441,395.898,172.337,37.945,157.181
C05170=1050.620,279.689,395.866,172.340,37.949,157.182
C05171=1050.626,279.937,395.836,172.344,37.952,157.183
C05172=1050.633,280.185,395.804,172.346,37.955,157.184
C05173=1050.639,280.433,395.774,172.349,37.959,157.185
C05174=1050.646,280.681,395.742,172.352,37.961,157.185
C05175=1050.652,280.928,395.711,172.355,37.965,157.186
C05176=1050.658,281.177,395.681,172.359,37.968,157.187
C05177=1050.665,281.425,395.649,172.361,37.971,157.187
C05178=1050.671,281.672,395.619,172.364,37.975,157.188
C05179=1050.678,281.920,395.587,172.367,37.978,157.189
C05180=1050.684,282.168,395.556,172.370,37.981,157.190
C05181=1050.691,282.417,395.525,172.374,37.984,157.191
C05182=1050.697,282.665,395.494,172.376,37.988,157.191
C05183=1050.704,282.912,395.463,172.380,37.991,157.192
C05184=1050.710,283.160,395.432,172.382,37.994,157.193
C05185=1050.717,283.408,395.401,172.386,37.997,157.194
C05186=1050.723,283.657,395.369,172.389,38.000,157.194
C05187=1050.729,283.904,395.337,172.391,38.004,157.195
C05188=1050.735,284.152,395.307,172.395,38.007,157.196
C05189=1050.742,284.400,395.275,172.397,38.010,157.197
C05190=1050.749,284.648,395.244,172.401,38.014,157.197
C05191=1050.755,284.896,395.212,172.404,38.016,157.198
C05192=1050.762,285.144,395.181,172.407,38.020,157.199
C05193=1050.769,285.392,395.150,172.410,38.023,157.200
C05194=1050.775,285.640,395.119,172.413,38.026,157.200
C05195=1050.781,285.887,395.088,172.416,38.030,157.201
C05196=1050.788,286.135,395.056,172.420,38.033,157.202
C05197=1050.795,286.383,395.025,172.422,38.036,157.203
C05198=1050.802,286.631,394.993,172.426,38.039,157.203
C05199=1050.808,286.879,394.962,172.429,38.043,157.204
C05200=1050.815,287.127,394.931,172.432,38.045,157.205
C05201=1050.822,287.375,394.899,172.435,38.049,157.206
C05202=1050.828,287.623,394.868,172.438,38.052,157.207
C05203=1050.834,287.871,394.836,172.441,38.055,157.207
C05204=1050.841,288.119,394.804,172.445,38.059,157.208
C05205=1050.848,288.367,394.773,172.447,38.062,157.209
C05206=1050.854,288.614,394.742,172.451,38.065,157.210
C05207=1050.860,288.862,394.710,172.455,38.069,157.210
C05208=1050.867,289.110,394.678,172.457,38.072,157.211
C05209=1050.873,289.358,394.647,172.461,38.075,157.212
C05210=1050.880,289.606,394.615,172.463,38.079,157.213
C05211=1050.886,289.854,394.583,172.467,38.082,157.214
C05212=1050.893,290.101,394.551,172.470,38.085,157.214
C05213=1050.900,290.369,394.518,172.473,38.089,157.215
C05214=1050.907,290.636,394.484,172.477,38.092,157.216
C05215=1050.915,290.904,394.450,172.480,38.096,157.217
C05216=1050.921,291.171,394.415,172.484,38.100,157.218
C05217=1050.928,291.419,394.384,172.487,38.103,157.218
C05218=1050.934,291.666,394.351,172.490,38.106,157.219
C05219=1050.941,291.914,394.319,172.493,38.109,157.220
C05220=1050.948,292.162,394.288,172.496,38.113,157.221
C05221=1050.954,292.410,394.255,172.500,38.116,157.222
C05222=1050.961,292.658,394.224,172.503,38.120,157.222
C05223=1050.967,292.906,394.192,172.506,38.122,157.223
C05224=1050.974,293.153,394.160,172.510,38.126,157.224
C05225=1050.980,293.401,394.128,172.512,38.129,157.225
C05226=1050.986,293.649,394.096,172.516,38.133,157.226
C05227=1050.994,293.897,394.064,172.520,38.136,157.226
C05228=1051.001,294.145,394.032,172.522,38.140,157.227
C05229=1051.007,294.393,394.000,172.526,38.143,157.228
C05230=1051.014,294.641,393.968,172.528,38.146,157.229
C05231=1051.020,294.889,393.936,172.532,38.149,157.230
C05232=1051.027,295.136,393.904,172.536,38.153,157.230
C05233=1051.033,295.384,393.872,172.538,38.156,157.231
C05234=1051.040,295.632,393.840,172.542,38.159,157.232
C05235=1051.046,295.880,393.808,172.546,38.163,157.233
C05236=1051.053,296.127,393.776,172.548,38.166,157.234
C05237=1051.059,296.375,393.744,172.552,38.170,157.234
C05238=1051.065,296.623,393.711,172.555,38.173,157.235
C05239=1051.072,296.870,393.679,172.558,38.176,157.236
C05240=1051.079,297.119,393.646,172.562,38.180,157.237
C05241=1051.085,297.367,393.613,172.565,38.183,157.238
C05242=1051.091,297.614,393.581,172.568,38.187,157.238
C05243=1051.097,297.863,393.549,172.572,38.191,157.239
C05244=1051.104,298.110,393.517,172.575,38.194,157.240
C05245=1051.111,298.357,393.484,172.579,38.197,157.241
C05246=1051.117,298.605,393.451,172.581,38.201,157.242
C05247=1051.123,298.853,393.419,172.585,38.204,157.243
C05248=1051.130,299.101,393.387,172.589,38.208,157.243
C05249=1051.136,299.348,393.354,172.591,38.211,157.244
C05250=1051.143,299.596,393.321,172.595,38.214,157.245
C05251=1051.149,299.844,393.288,172.599,38.218,157.246
C05252=1051.155,300.092,393.256,172.601,38.222,157.247
C05253=1051.162,300.340,393.224,172.605,38.225,157.248
C05254=1051.169,300.587,393.191,172.609,38.229,157.249
C05255=1051.175,300.835,393.159,172.611,38.232,157.249
C05256=1051.182,301.083,393.126,172.615,38.235,157.250
C05257=1051.188,301.331,393.093,172.619,38.239,157.251
C05258=1051.195,301.578,393.060,172.622,38.242,157.252
C05259=1051.202,301.825,393.028,172.625,38.246,157.253
C05260=1051.208,302.073,392.995,172.629,38.250,157.254
C05261=1051.215,302.321,392.962,172.633,38.253,157.254
C05262=1051.221,302.569,392.929,172.635,38.256,157.255
C05263=1051.227,302.817,392.897,172.639,38.260,157.256
C05264=1051.234,303.064,392.864,172.643,38.263,157.257
C05265=1051.241,303.312,392.831,172.645,38.267,157.258
C05266=1051.248,303.560,392.799,172.649,38.270,157.259
C05267=1051.254,303.807,392.766,172.653,38.274,157.259
C05268=1051.261,304.056,392.733,172.657,38.277,157.260
C05269=1051.268,304.338,392.696,172.660,38.281,157.261
C05270=1051.276,304.621,392.658,172.664,38.285,157.262
C05271=1051.283,304.905,392.620,172.668,38.289,157.263
C05272=1051.291,305.188,392.582,172.672,38.293,157.264
C05273=1051.297,305.436,392.549,172.676,38.297,157.265
C05274=1051.304,305.684,392.517,172.679,38.300,157.266
C05275=1051.311,305.931,392.484,172.683,38.304,157.267
C05276=1051.318,306.180,392.451,172.686,38.307,157.268
C05277=1051.324,306.427,392.418,172.689,38.311,157.268
C05278=1051.331,306.674,392.385,172.693,38.314,157.269
C05279=1051.337,306.922,392.352,172.697,38.318,157.270
C05280=1051.344,307.170,392.319,172.700,38.321,157.271
C05281=1051.351,307.418,392.285,172.703,38.325,157.272
C05282=1051.357,307.665,392.253,172.707,38.329,157.273
C05283=1051.364,307.913,392.221,172.711,38.332,157.274
C05284=1051.371,308.160,392.187,172.714,38.335,157.274
C05285=1051.378,308.408,392.154,172.718,38.339,157.275
C05286=1051.385,308.656,392.121,172.721,38.343,157.276
C05287=1051.391,308.903,392.087,172.725,38.346,157.277
C05288=1051.398,309.151,392.054,172.728,38.349,157.278
C05289=1051.405,309.398,392.021,172.732,38.353,157.279
C05290=1051.412,309.647,391.988,172.736,38.357,157.280
C05291=1051.418,309.894,391.955,172.739,38.360,157.280
C05292=1051.425,310.142,391.921,172.743,38.364,157.281
C05293=1051.431,310.390,391.888,172.746,38.367,157.282
C05294=1051.439,310.637,391.855,172.750,38.371,157.283
C05295=1051.446,310.885,391.822,172.753,38.374,157.284
C05296=1051.453,311.132,391.789,172.757,38.378,157.285
C05297=1051.460,311.381,391.756,172.761,38.381,157.286
C05298=1051.466,311.627,391.722,172.765,38.385,157.286
C05299=1051.473,311.876,391.689,172.768,38.389,157.287
C05300=1051.480,312.123,391.656,172.772,38.392,157.288
C05301=1051.487,312.370,391.622,172.775,38.396,157.289
C05302=1051.494,312.619,391.589,172.779,38.399,157.290
C05303=1051.500,312.866,391.555,172.782,38.403,157.291
C05304=1051.507,313.114,391.522,172.786,38.407,157.292
C05305=1051.513,313.361,391.488,172.790,38.410,157.293
C05306=1051.520,313.609,391.454,172.794,38.414,157.294
C05307=1051.527,313.856,391.421,172.797,38.418,157.295
C05308=1051.533,314.105,391.387,172.801,38.421,157.295
C05309=1051.540,314.351,391.354,172.804,38.425,157.296
C05310=1051.546,314.599,391.319,172.808,38.428,157.297
C05311=1051.553,314.847,391.285,172.812,38.432,157.298
C05312=1051.559,315.094,391.251,172.815,38.436,157.299
C05313=1051.567,315.342,391.217,172.819,38.440,157.300
C05314=1051.572,315.589,391.183,172.823,38.444,157.301
C05315=1051.580,315.837,391.150,172.827,38.447,157.302
C05316=1051.585,316.084,391.115,172.831,38.451,157.303
C05317=1051.593,316.332,391.082,172.834,38.455,157.304
C05318=1051.599,316.580,391.047,172.837,38.459,157.305
C05319=1051.606,316.827,391.014,172.841,38.463,157.306
C05320=1051.612,317.075,390.979,172.845,38.466,157.306
C05321=1051.619,317.323,390.946,172.848,38.470,157.307
C05322=1051.625,317.570,390.911,172.852,38.474,157.308
C05323=1051.632,317.818,390.878,172.856,38.478,157.309
C05324=1051.639,318.066,390.843,172.860,38.481,157.310
C05325=1051.646,318.354,390.804,172.864,38.486,157.311
C05326=1051.654,318.640,390.765,172.869,38.490,157.312
C05327=1051.661,318.928,390.725,172.873,38.495,157.313
C05328=1051.669,319.216,390.685,172.878,38.499,157.315
C05329=1051.676,319.463,390.651,172.881,38.503,157.316
C05330=1051.683,319.711,390.616,172.885,38.506,157.316
C05331=1051.690,319.959,390.583,172.889,38.510,157.317
C05332=1051.696,320.206,390.549,172.893,38.514,157.318
C05333=1051.704,320.453,390.514,172.897,38.518,157.319
C05334=1051.710,320.701,390.480,172.900,38.522,157.320
C05335=1051.717,320.949,390.446,172.904,38.525,157.321
C05336=1051.723,321.196,390.412,172.908,38.529,157.322
C05337=1051.730,321.444,390.377,172.912,38.533,157.323
C05338=1051.737,321.691,390.343,172.916,38.537,157.324
C05339=1051.743,321.939,390.308,172.920,38.541,157.325
C05340=1051.751,322.186,390.274,172.923,38.545,157.326
C05341=1051.757,322.434,390.239,172.927,38.549,157.327
C05342=1051.764,322.682,390.205,172.931,38.552,157.328
C05343=1051.771,322.929,390.171,172.935,38.556,157.329
C05344=1051.777,323.177,390.136,172.939,38.560,157.330
C05345=1051.785,323.424,390.102,172.943,38.564,157.331
C05346=1051.791,323.672,390.067,172.946,38.568,157.332
C05347=1051.798,323.920,390.034,172.950,38.571,157.333
C05348=1051.805,324.167,389.998,172.954,38.575,157.334
C05349=1051.812,324.415,389.964,172.958,38.579,157.335
C05350=1051.819,324.662,389.930,172.962,38.583,157.336
C05351=1051.826,324.910,389.895,172.966,38.587,157.337
C05352=1051.832,325.157,389.860,172.969,38.591,157.338
C05353=1051.840,325.405,389.826,172.973,38.595,157.338
C05354=1051.846,325.652,389.791,172.977,38.599,157.339
C05355=1051.854,325.899,389.756,172.981,38.603,157.340
C05356=1051.860,326.147,389.722,172.985,38.606,157.341
C05357=1051.867,326.395,389.687,172.990,38.610,157.342
C05358=1051.874,326.642,389.653,172.994,38.614,157.343
C05359=1051.881,326.890,389.618,172.997,38.618,157.344
C05360=1051.888,327.137,389.583,173.001,38.622,157.345
C05361=1051.895,327.385,389.549,173.005,38.626,157.346
C05362=1051.902,327.632,389.514,173.009,38.630,157.347
C05363=1051.909,327.879,389.479,173.013,38.634,157.348
C05364=1051.916,328.127,389.444,173.017,38.638,157.349
C05365=1051.923,328.375,389.410,173.022,38.641,157.350
C05366=1051.930,328.622,389.375,173.025,38.645,157.351
C05367=1051.937,328.870,389.340,173.029,38.649,157.352
C05368=1051.944,329.117,389.305,173.033,38.653,157.353
C05369=1051.952,329.364,389.270,173.037,38.657,157.354
C05370=1051.958,329.612,389.236,173.041,38.661,157.355
C05371=1051.965,329.859,389.200,173.046,38.665,157.356
C05372=1051.972,330.107,389.165,173.050,38.669,157.357
C05373=1051.978,330.354,389.130,173.054,38.673,157.358
C05374=1051.985,330.602,389.095,173.057,38.677,157.359
C05375=1051.993,330.850,389.060,173.061,38.681,157.360
C05376=1051.999,331.097,389.024,173.065,38.685,157.361
C05377=1052.006,331.344,388.989,173.069,38.689,157.362
C05378=1052.013,331.592,388.954,173.074,38.693,157.363
C05379=1052.020,331.839,388.919,173.078,38.697,157.364
C05380=1052.027,332.086,388.883,173.082,38.702,157.365
C05381=1052.034,332.369,388.842,173.087,38.706,157.367
C05382=1052.042,332.651,388.802,173.091,38.711,157.368
C05383=1052.051,332.933,388.762,173.096,38.716,157.369
C05384=1052.058,333.216,388.722,173.100,38.720,157.370
C05385=1052.065,333.464,388.686,173.105,38.724,157.371
C05386=1052.072,333.711,388.651,173.109,38.728,157.372
C05387=1052.079,333.959,388.616,173.113,38.733,157.373
C05388=1052.086,334.205,388.580,173.117,38.737,157.374
C05389=1052.093,334.453,388.545,173.122,38.741,157.375
C05390=1052.100,334.701,388.509,173.126,38.745,157.376
C05391=1052.107,334.948,388.474,173.130,38.749,157.378
C05392=1052.114,335.195,388.438,173.134,38.753,157.379
C05393=1052.121,335.443,388.403,173.139,38.757,157.380
C05394=1052.127,335.691,388.367,173.142,38.761,157.381
C05395=1052.134,335.937,388.331,173.146,38.766,157.382
C05396=1052.141,336.185,388.296,173.150,38.770,157.383
C05397=1052.149,336.432,388.260,173.155,38.774,157.384
C05398=1052.155,336.680,388.225,173.159,38.778,157.385
C05399=1052.162,336.927,388.188,173.163,38.782,157.386
C05400=1052.169,337.175,388.153,173.167,38.787,157.387
C05401=1052.176,337.421,388.117,173.172,38.791,157.388
C05402=1052.183,337.669,388.082,173.176,38.795,157.389
C05403=1052.190,337.917,388.045,173.180,38.799,157.390
C05404=1052.197,338.163,388.009,173.184,38.804,157.391
C05405=1052.204,338.411,387.974,173.189,38.808,157.393
C05406=1052.211,338.658,387.937,173.193,38.812,157.394
C05407=1052.217,338.906,387.902,173.197,38.816,157.395
C05408=1052.225,339.153,387.866,173.202,38.821,157.396
C05409=1052.231,339.400,387.830,173.206,38.825,157.397
C05410=1052.238,339.647,387.794,173.210,38.830,157.398
C05411=1052.245,339.895,387.758,173.215,38.833,157.399
C05412=1052.252,340.142,387.722,173.219,38.838,157.400
C05413=1052.260,340.390,387.686,173.223,38.842,157.401
C05414=1052.266,340.637,387.649,173.228,38.847,157.402
C05415=1052.274,340.885,387.614,173.232,38.851,157.404
C05416=1052.281,341.131,387.578,173.236,38.855,157.405
C05417=1052.288,341.379,387.541,173.241,38.860,157.406
C05418=1052.295,341.626,387.505,173.245,38.864,157.407
C05419=1052.302,341.873,387.469,173.249,38.868,157.408
C05420=1052.309,342.120,387.432,173.254,38.872,157.409
C05421=1052.316,342.368,387.396,173.258,38.877,157.410
C05422=1052.322,342.616,387.360,173.262,38.881,157.411
C05423=1052.330,342.863,387.324,173.267,38.886,157.413
C05424=1052.337,343.109,387.287,173.271,38.890,157.414
C05425=1052.344,343.357,387.251,173.276,38.894,157.415
C05426=1052.351,343.604,387.214,173.280,38.899,157.416
C05427=1052.358,343.851,387.178,173.284,38.904,157.417
C05428=1052.365,344.098,387.142,173.289,38.908,157.418
C05429=1052.372,344.346,387.106,173.293,38.913,157.419
C05430=1052.379,344.593,387.069,173.298,38.917,157.421
C05431=1052.386,344.841,387.032,173.302,38.921,157.422
C05432=1052.393,345.088,386.996,173.306,38.926,157.423
C05433=1052.400,345.335,386.959,173.312,38.931,157.424
C05434=1052.407,345.582,386.922,173.316,38.935,157.425
C05435=1052.414,345.829,386.886,173.321,38.939,157.426
C05436=1052.421,346.077,386.849,173.325,38.944,157.428
C05437=1052.429,346.355,386.808,173.330,38.949,157.429
C05438=1052.437,346.633,386.767,173.335,38.954,157.430
C05439=1052.444,346.912,386.725,173.340,38.959,157.432
C05440=1052.454,347.190,386.684,173.346,38.964,157.433
C05441=1052.460,347.437,386.647,173.350,38.969,157.434
C05442=1052.467,347.685,386.610,173.355,38.973,157.435
C05443=1052.474,347.932,386.573,173.359,38.978,157.437
C05444=1052.481,348.179,386.537,173.364,38.982,157.438
C05445=1052.489,348.426,386.499,173.368,38.987,157.439
C05446=1052.495,348.674,386.463,173.373,38.992,157.440
C05447=1052.503,348.920,386.426,173.377,38.996,157.441
C05448=1052.510,349.168,386.389,173.382,39.001,157.443
C05449=1052.517,349.415,386.352,173.386,39.005,157.444
C05450=1052.524,349.663,386.315,173.391,39.010,157.445
C05451=1052.532,349.910,386.278,173.396,39.015,157.446
C05452=1052.539,350.156,386.241,173.401,39.019,157.447
C05453=1052.545,350.404,386.204,173.405,39.024,157.449
C05454=1052.553,350.651,386.166,173.410,39.028,157.450
C05455=1052.561,350.898,386.130,173.414,39.033,157.451
C05456=1052.568,351.145,386.093,173.419,39.038,157.452
C05457=1052.574,351.392,386.056,173.423,39.043,157.453
